C08939=1023.663,350.015,-141.631,171.610,48.646,159.588
C08940=1023.670,350.262,-141.669,171.618,48.645,159.589
C08941=1023.678,350.509,-141.706,171.625,48.645,159.590
C08942=1023.686,350.757,-141.744,171.632,48.644,159.591
C08943=1023.693,350.988,-141.779,171.639,48.644,159.591
C08944=1023.700,351.219,-141.813,171.645,48.643,159.592
C08945=1023.707,351.450,-141.849,171.651,48.643,159.593
C08946=1023.714,351.682,-141.884,171.658,48.643,159.594
C08947=1023.722,351.913,-141.919,171.665,48.642,159.595
C08948=1023.729,352.145,-141.954,171.671,48.642,159.596
C08949=1023.736,352.376,-141.990,171.678,48.641,159.597
C08950=1023.744,352.607,-142.025,171.685,48.641,159.598
C08951=1023.752,352.855,-142.063,171.692,48.640,159.598
C08952=1023.759,353.101,-142.101,171.699,48.640,159.599
C08953=1023.767,353.348,-142.138,171.706,48.640,159.600
C08954=1023.775,353.595,-142.177,171.713,48.639,159.601
C08955=1023.783,353.843,-142.214,171.721,48.639,159.602
C08956=1023.792,354.089,-142.252,171.727,48.638,159.603
C08957=1023.799,354.337,-142.290,171.735,48.638,159.604
C08958=1023.806,354.583,-142.328,171.742,48.638,159.605
C08959=1023.814,354.831,-142.366,171.749,48.637,159.606
C08960=1023.823,355.077,-142.404,171.757,48.637,159.607
C08961=1023.831,355.324,-142.442,171.764,48.637,159.608
C08962=1023.838,355.572,-142.480,171.771,48.636,159.609
C08963=1023.846,355.819,-142.518,171.779,48.636,159.610
C08964=1023.854,356.065,-142.557,171.786,48.636,159.611
C08965=1023.861,356.312,-142.595,171.793,48.636,159.612
C08966=1023.869,356.560,-142.633,171.801,48.635,159.613
C08967=1023.877,356.806,-142.670,171.808,48.635,159.614
C08968=1023.885,357.053,-142.709,171.815,48.634,159.615
C08969=1023.894,357.300,-142.748,171.823,48.634,159.616
C08970=1023.901,357.547,-142.786,171.830,48.634,159.617
C08971=1023.909,357.794,-142.824,171.837,48.634,159.618
C08972=1023.917,358.040,-142.863,171.845,48.634,159.619
C08973=1023.925,358.288,-142.901,171.852,48.634,159.620
C08974=1023.933,358.535,-142.940,171.860,48.633,159.622
C08975=1023.941,358.781,-142.978,171.867,48.633,159.623
C08976=1023.950,359.028,-143.016,171.874,48.633,159.624
C08977=1023.957,359.275,-143.054,171.883,48.633,159.625
C08978=1023.965,359.522,-143.093,171.890,48.633,159.626
C08979=1023.973,359.769,-143.132,171.898,48.633,159.627
C08980=1023.981,360.016,-143.170,171.905,48.632,159.628
C08981=1023.989,360.262,-143.209,171.912,48.632,159.629
C08982=1023.998,360.510,-143.248,171.920,48.632,159.630
C08983=1024.005,360.757,-143.287,171.927,48.632,159.631
C08984=1024.013,361.003,-143.326,171.935,48.632,159.632
C08985=1024.021,361.250,-143.365,171.942,48.632,159.633
C08986=1024.029,361.497,-143.403,171.950,48.632,159.634
C08987=1024.037,361.743,-143.442,171.958,48.632,159.636
C08988=1024.044,361.991,-143.481,171.966,48.632,159.637
C08989=1024.053,362.237,-143.521,171.973,48.632,159.638
C08990=1024.061,362.485,-143.559,171.981,48.632,159.639
C08991=1024.070,362.731,-143.599,171.988,48.632,159.640
C08992=1024.077,362.978,-143.637,171.997,48.632,159.641
C08993=1024.085,363.225,-143.677,172.004,48.633,159.643
C08994=1024.093,363.471,-143.716,172.012,48.632,159.644
C08995=1024.101,363.719,-143.755,172.019,48.633,159.645
C08996=1024.110,363.965,-143.794,172.027,48.632,159.646
C08997=1024.118,364.212,-143.833,172.035,48.633,159.647
C08998=1024.126,364.459,-143.873,172.043,48.633,159.648
C08999=1024.134,364.706,-143.912,172.050,48.633,159.650
C09000=1024.142,364.952,-143.951,172.058,48.633,159.651
C09001=1024.150,365.198,-143.990,172.066,48.633,159.652
C09002=1024.159,365.446,-144.029,172.074,48.634,159.653
C09003=1024.168,365.738,-144.076,172.084,48.633,159.655
C09004=1024.179,366.031,-144.123,172.093,48.633,159.656
C09005=1024.188,366.323,-144.169,172.103,48.634,159.657
C09006=1024.198,366.616,-144.216,172.111,48.634,159.659
C09007=1024.206,366.862,-144.256,172.120,48.634,159.660
C09008=1024.215,367.109,-144.295,172.128,48.635,159.661
C09009=1024.223,367.355,-144.334,172.136,48.635,159.663
C09010=1024.231,367.602,-144.374,172.144,48.635,159.664
C09011=1024.239,367.849,-144.413,172.152,48.635,159.665
C09012=1024.248,368.096,-144.453,172.159,48.636,159.666
C09013=1024.257,368.343,-144.492,172.168,48.636,159.668
C09014=1024.265,368.589,-144.533,172.176,48.636,159.669
C09015=1024.273,368.836,-144.572,172.184,48.637,159.670
C09016=1024.281,369.083,-144.612,172.192,48.637,159.671
C09017=1024.290,369.328,-144.652,172.200,48.637,159.673
C09018=1024.298,369.575,-144.692,172.208,48.638,159.674
C09019=1024.307,369.823,-144.732,172.216,48.638,159.675
C09020=1024.315,370.069,-144.773,172.225,48.638,159.676
C09021=1024.323,370.316,-144.812,172.232,48.639,159.678
C09022=1024.331,370.562,-144.853,172.241,48.640,159.679
C09023=1024.340,370.808,-144.892,172.249,48.640,159.681
C09024=1024.348,371.055,-144.933,172.258,48.640,159.682
C09025=1024.356,371.302,-144.973,172.265,48.641,159.683
C09026=1024.365,371.548,-145.013,172.274,48.641,159.685
C09027=1024.373,371.795,-145.054,172.282,48.642,159.686
C09028=1024.382,372.042,-145.093,172.291,48.642,159.687
C09029=1024.390,372.288,-145.134,172.299,48.643,159.689
C09030=1024.399,372.535,-145.174,172.307,48.643,159.690
C09031=1024.407,372.782,-145.214,172.316,48.644,159.691
C09032=1024.416,373.028,-145.254,172.324,48.644,159.693
C09033=1024.424,373.275,-145.295,172.333,48.645,159.694
C09034=1024.433,373.521,-145.335,172.341,48.645,159.695
C09035=1024.442,373.768,-145.376,172.349,48.646,159.697
C09036=1024.449,374.015,-145.416,172.357,48.647,159.698
C09037=1024.459,374.261,-145.457,172.366,48.647,159.700
C09038=1024.467,374.508,-145.497,172.375,48.648,159.701
C09039=1024.475,374.719,-145.532,172.382,48.648,159.702
C09040=1024.482,374.931,-145.567,172.389,48.649,159.703
C09041=1024.489,375.143,-145.602,172.397,48.649,159.705
C09042=1024.497,375.354,-145.637,172.404,48.650,159.706
C09043=1024.505,375.566,-145.671,172.412,48.650,159.707
C09044=1024.512,375.778,-145.706,172.419,48.651,159.708
C09045=1024.520,375.989,-145.741,172.426,48.651,159.710
C09046=1024.527,376.201,-145.776,172.434,48.652,159.711
C09047=1024.536,376.448,-145.817,172.443,48.653,159.712
C09048=1024.545,376.694,-145.858,172.451,48.653,159.714
C09049=1024.553,376.941,-145.899,172.459,48.655,159.715
C09050=1024.562,377.187,-145.939,172.468,48.655,159.717
C09051=1024.570,377.433,-145.981,172.477,48.656,159.718
C09052=1024.579,377.680,-146.022,172.485,48.657,159.720
C09053=1024.587,377.926,-146.063,172.494,48.658,159.721
C09054=1024.596,378.173,-146.104,172.503,48.659,159.723
C09055=1024.605,378.419,-146.146,172.512,48.659,159.724
C09056=1024.614,378.665,-146.186,172.520,48.660,159.726
C09057=1024.623,378.912,-146.228,172.529,48.661,159.727
C09058=1024.631,379.159,-146.269,172.538,48.662,159.729
C09059=1024.640,379.404,-146.310,172.547,48.663,159.730
C09060=1024.649,379.651,-146.352,172.555,48.663,159.732
C09061=1024.657,379.898,-146.393,172.565,48.665,159.734
C09062=1024.666,380.144,-146.435,172.574,48.665,159.735
C09063=1024.675,380.389,-146.475,172.583,48.666,159.737
C09064=1024.684,380.635,-146.517,172.592,48.667,159.738
C09065=1024.692,380.880,-146.559,172.601,48.668,159.740
C09066=1024.702,381.126,-146.600,172.610,48.669,159.741
C09067=1024.710,381.372,-146.641,172.618,48.670,159.743
C09068=1024.719,381.617,-146.682,172.628,48.671,159.745
C09069=1024.728,381.862,-146.724,172.636,48.672,159.746
C09070=1024.737,382.109,-146.766,172.645,48.673,159.748
C09071=1024.746,382.355,-146.807,172.654,48.674,159.749
C09072=1024.755,382.601,-146.849,172.664,48.675,159.751
C09073=1024.764,382.847,-146.890,172.673,48.676,159.753
C09074=1024.773,383.094,-146.932,172.682,48.677,159.754
C09075=1024.782,383.340,-146.974,172.691,48.678,159.756
C09076=1024.791,383.586,-147.015,172.700,48.680,159.757
C09077=1024.800,383.832,-147.058,172.710,48.680,159.759
C09078=1024.809,384.079,-147.100,172.719,48.681,159.761
C09079=1024.818,384.325,-147.141,172.728,48.683,159.762
C09080=1024.827,384.571,-147.183,172.738,48.684,159.764
C09081=1024.837,384.817,-147.225,172.747,48.685,159.766
C09082=1024.846,385.063,-147.267,172.756,48.686,159.767
C09083=1024.856,385.310,-147.309,172.765,48.687,159.769
C09084=1024.865,385.556,-147.351,172.775,48.688,159.771
C09085=1024.874,385.802,-147.393,172.784,48.690,159.773
C09086=1024.883,386.049,-147.435,172.793,48.691,159.774
C09087=1024.892,386.294,-147.477,172.803,48.692,159.776
C09088=1024.902,386.541,-147.520,172.812,48.693,159.778
C09089=1024.911,386.787,-147.561,172.822,48.695,159.780
C09090=1024.919,387.033,-147.605,172.832,48.696,159.781
C09091=1024.929,387.279,-147.647,172.841,48.697,159.783
C09092=1024.938,387.526,-147.689,172.851,48.698,159.785
C09093=1024.947,387.772,-147.731,172.860,48.700,159.786
C09094=1024.957,388.018,-147.774,172.869,48.701,159.788
C09095=1024.966,388.264,-147.817,172.880,48.702,159.790
C09096=1024.975,388.510,-147.860,172.889,48.704,159.792
C09097=1024.984,388.756,-147.902,172.899,48.705,159.794
C09098=1024.994,389.002,-147.945,172.908,48.706,159.795
C09099=1025.003,389.248,-147.987,172.919,48.708,159.797
C09100=1025.012,389.495,-148.031,172.928,48.709,159.799
C09101=1025.022,389.740,-148.073,172.938,48.710,159.801
C09102=1025.031,389.986,-148.116,172.947,48.712,159.803
C09103=1025.041,390.233,-148.158,172.958,48.713,159.805
C09104=1025.049,390.479,-148.201,172.967,48.715,159.806
C09105=1025.059,390.725,-148.244,172.977,48.716,159.808
C09106=1025.068,390.970,-148.287,172.987,48.718,159.810
C09107=1025.078,391.217,-148.331,172.997,48.720,159.812
C09108=1025.087,391.463,-148.373,173.006,48.721,159.814
C09109=1025.097,391.709,-148.417,173.017,48.723,159.816
C09110=1025.106,391.955,-148.460,173.026,48.725,159.818
C09111=1025.115,392.201,-148.503,173.036,48.726,159.820
C09112=1025.125,392.447,-148.546,173.047,48.727,159.821
C09113=1025.135,392.694,-148.589,173.056,48.729,159.823
C09114=1025.144,392.939,-148.633,173.067,48.731,159.825
C09115=1025.154,393.185,-148.675,173.077,48.732,159.827
C09116=1025.163,393.431,-148.720,173.087,48.734,159.829
C09117=1025.173,393.677,-148.763,173.097,48.736,159.831
C09118=1025.182,393.923,-148.806,173.108,48.738,159.833
C09119=1025.192,394.169,-148.850,173.117,48.739,159.835
C09120=1025.202,394.415,-148.894,173.128,48.741,159.837
C09121=1025.211,394.660,-148.937,173.138,48.743,159.839
C09122=1025.221,394.906,-148.981,173.147,48.745,159.841
C09123=1025.232,395.188,-149.030,173.159,48.746,159.843
C09124=1025.242,395.469,-149.081,173.171,48.748,159.846
C09125=1025.254,395.750,-149.131,173.183,48.751,159.848
C09126=1025.265,396.031,-149.181,173.195,48.753,159.850
C09127=1025.274,396.277,-149.225,173.206,48.754,159.852
C09128=1025.284,396.523,-149.268,173.216,48.756,159.855
C09129=1025.294,396.769,-149.312,173.227,48.758,159.856
C09130=1025.304,397.015,-149.356,173.236,48.760,159.858
C09131=1025.313,397.261,-149.400,173.247,48.762,159.861
C09132=1025.324,397.507,-149.444,173.258,48.763,159.863
C09133=1025.333,397.752,-149.488,173.269,48.766,159.865
C09134=1025.343,397.998,-149.532,173.279,48.767,159.867
C09135=1025.353,398.244,-149.576,173.290,48.769,159.869
C09136=1025.363,398.490,-149.621,173.301,48.771,159.871
C09137=1025.373,398.735,-149.664,173.311,48.773,159.873
C09138=1025.383,398.982,-149.709,173.322,48.775,159.875
C09139=1025.392,399.228,-149.754,173.333,48.777,159.878
C09140=1025.403,399.473,-149.798,173.343,48.779,159.880
C09141=1025.412,399.719,-149.842,173.354,48.781,159.882
C09142=1025.422,399.965,-149.887,173.365,48.783,159.884
C09143=1025.432,400.210,-149.932,173.376,48.785,159.886
C09144=1025.443,400.456,-149.976,173.387,48.787,159.888
C09145=1025.452,400.702,-150.020,173.397,48.789,159.891
C09146=1025.462,400.948,-150.065,173.408,48.792,159.893
C09147=1025.472,401.193,-150.110,173.419,48.794,159.895
C09148=1025.483,401.439,-150.155,173.430,48.796,159.897
C09149=1025.492,401.685,-150.199,173.441,48.798,159.899
C09150=1025.502,401.930,-150.244,173.452,48.800,159.902
C09151=1025.512,402.176,-150.289,173.463,48.803,159.904
C09152=1025.522,402.422,-150.334,173.475,48.804,159.906
C09153=1025.532,402.667,-150.379,173.485,48.807,159.908
C09154=1025.542,402.914,-150.424,173.497,48.809,159.911
C09155=1025.552,403.159,-150.470,173.508,48.811,159.913
C09156=1025.562,403.405,-150.515,173.518,48.813,159.915
C09157=1025.572,403.650,-150.560,173.531,48.816,159.918
C09158=1025.582,403.896,-150.605,173.541,48.818,159.920
C09159=1025.593,404.141,-150.650,173.553,48.821,159.922
C09160=1025.604,404.387,-150.695,173.563,48.823,159.924
C09161=1025.614,404.632,-150.741,173.576,48.825,159.927
C09162=1025.624,404.878,-150.786,173.586,48.827,159.929
C09163=1025.634,405.123,-150.831,173.598,48.830,159.932
C09164=1025.644,405.369,-150.877,173.610,48.832,159.934
C09165=1025.655,405.615,-150.922,173.621,48.835,159.936
C09166=1025.665,405.861,-150.967,173.632,48.837,159.939
C09167=1025.675,406.106,-151.013,173.644,48.839,159.941
C09168=1025.686,406.352,-151.059,173.655,48.842,159.944
C09169=1025.696,406.597,-151.104,173.668,48.844,159.946
C09170=1025.706,406.843,-151.150,173.679,48.847,159.948
C09171=1025.717,407.088,-151.196,173.690,48.850,159.951
C09172=1025.727,407.334,-151.242,173.702,48.852,159.953
C09173=1025.738,407.580,-151.288,173.713,48.854,159.956
C09174=1025.749,407.825,-151.333,173.726,48.857,159.958
C09175=1025.759,408.070,-151.379,173.738,48.859,159.961
C09176=1025.770,408.315,-151.424,173.749,48.862,159.963
C09177=1025.781,408.561,-151.470,173.761,48.864,159.966
C09178=1025.791,408.807,-151.516,173.772,48.867,159.968
C09179=1025.802,409.052,-151.562,173.785,48.870,159.971
C09180=1025.813,409.299,-151.608,173.796,48.872,159.973
C09181=1025.824,409.544,-151.654,173.808,48.874,159.976
C09182=1025.834,409.790,-151.700,173.821,48.877,159.978
C09183=1025.847,410.093,-151.758,173.835,48.881,159.981
C09184=1025.860,410.397,-151.815,173.850,48.884,159.985
C09185=1025.874,410.700,-151.872,173.865,48.887,159.988
C09186=1025.887,411.004,-151.931,173.881,48.891,159.991
C09187=1025.897,411.250,-151.977,173.893,48.893,159.994
C09188=1025.909,411.495,-152.023,173.905,48.897,159.996
C09189=1025.919,411.741,-152.070,173.917,48.899,159.999
C09190=1025.929,411.986,-152.117,173.930,48.902,160.002
C09191=1025.940,412.231,-152.163,173.942,48.905,160.004
C09192=1025.951,412.476,-152.210,173.954,48.908,160.007
C09193=1025.962,412.722,-152.257,173.966,48.911,160.010
C09194=1025.973,412.968,-152.303,173.979,48.913,160.012
C09195=1025.984,413.213,-152.350,173.991,48.916,160.015
C09196=1025.995,413.458,-152.397,174.004,48.919,160.018
C09197=1026.005,413.704,-152.444,174.017,48.922,160.020
C09198=1026.017,413.949,-152.491,174.029,48.925,160.023
C09199=1026.028,414.194,-152.538,174.042,48.928,160.026
C09200=1026.039,414.440,-152.586,174.055,48.931,160.029
C09201=1026.050,414.685,-152.633,174.067,48.934,160.031
C09202=1026.061,414.930,-152.680,174.080,48.936,160.034
C09203=1026.072,415.175,-152.726,174.093,48.940,160.037
C09204=1026.083,415.421,-152.774,174.105,48.943,160.040
C09205=1026.094,415.666,-152.821,174.118,48.946,160.043
C09206=1026.106,415.911,-152.868,174.131,48.949,160.045
C09207=1026.117,416.157,-152.917,174.145,48.952,160.048
C09208=1026.128,416.402,-152.963,174.157,48.955,160.051
C09209=1026.139,416.647,-153.011,174.170,48.958,160.054
C09210=1026.150,416.891,-153.059,174.183,48.961,160.057
C09211=1026.161,417.137,-153.106,174.196,48.965,160.060
C09212=1026.173,417.382,-153.154,174.209,48.967,160.062
C09213=1026.184,417.628,-153.202,174.223,48.970,160.065
C09214=1026.195,417.872,-153.250,174.236,48.974,160.068
C09215=1026.206,418.118,-153.297,174.249,48.977,160.071
C09216=1026.217,418.363,-153.346,174.262,48.980,160.074
C09217=1026.229,418.608,-153.393,174.275,48.983,160.077
C09218=1026.240,418.854,-153.442,174.288,48.987,160.080
C09219=1026.252,419.099,-153.489,174.303,48.990,160.083
C09220=1026.263,419.344,-153.538,174.316,48.994,160.086
C09221=1026.275,419.589,-153.586,174.329,48.997,160.089
C09222=1026.286,419.834,-153.634,174.343,49.000,160.092
C09223=1026.298,420.079,-153.682,174.356,49.004,160.095
C09224=1026.309,420.324,-153.730,174.370,49.007,160.098
C09225=1026.321,420.569,-153.779,174.383,49.011,160.101
C09226=1026.332,420.814,-153.827,174.397,49.014,160.104
C09227=1026.344,421.059,-153.875,174.411,49.017,160.107
C09228=1026.356,421.304,-153.924,174.424,49.020,160.110
C09229=1026.367,421.549,-153.972,174.439,49.024,160.114
C09230=1026.379,421.794,-154.020,174.452,49.027,160.117
C09231=1026.391,422.039,-154.070,174.466,49.031,160.120
C09232=1026.403,422.284,-154.118,174.480,49.034,160.123
C09233=1026.414,422.529,-154.167,174.494,49.038,160.126
C09234=1026.426,422.774,-154.216,174.508,49.042,160.129
C09235=1026.438,423.019,-154.265,174.522,49.045,160.132
C09236=1026.450,423.264,-154.313,174.536,49.049,160.136
C09237=1026.461,423.508,-154.362,174.550,49.052,160.139
C09238=1026.473,423.754,-154.412,174.564,49.056,160.142
C09239=1026.485,423.999,-154.461,174.578,49.059,160.145
C09240=1026.497,424.244,-154.510,174.593,49.063,160.148
C09241=1026.509,424.488,-154.559,174.607,49.067,160.152
C09242=1026.521,424.734,-154.608,174.622,49.070,160.155
C09243=1026.536,425.048,-154.672,174.641,49.075,160.159
C09244=1026.551,425.362,-154.735,174.658,49.080,160.164
C09245=1026.567,425.676,-154.798,174.677,49.085,160.168
C09246=1026.582,425.990,-154.861,174.696,49.090,160.172
C09247=1026.594,426.236,-154.911,174.711,49.094,160.175
C09248=1026.607,426.480,-154.961,174.725,49.098,160.179
C09249=1026.618,426.725,-155.010,174.740,49.101,160.182
C09250=1026.630,426.970,-155.060,174.755,49.105,160.186
C09251=1026.643,427.215,-155.110,174.770,49.109,160.189
C09252=1026.655,427.460,-155.160,174.785,49.113,160.192
C09253=1026.667,427.704,-155.210,174.799,49.117,160.196
C09254=1026.679,427.949,-155.260,174.814,49.121,160.199
C09255=1026.691,428.193,-155.310,174.830,49.124,160.203
C09256=1026.704,428.438,-155.360,174.845,49.128,160.206
C09257=1026.716,428.683,-155.410,174.860,49.133,160.210
C09258=1026.728,428.928,-155.460,174.875,49.136,160.213
C09259=1026.740,429.172,-155.510,174.890,49.140,160.217
C09260=1026.752,429.417,-155.560,174.905,49.145,160.220
C09261=1026.765,429.661,-155.611,174.921,49.148,160.224
C09262=1026.777,429.906,-155.661,174.936,49.153,160.228
C09263=1026.790,430.151,-155.712,174.952,49.156,160.231
C09264=1026.803,430.396,-155.762,174.967,49.161,160.235
C09265=1026.815,430.640,-155.813,174.983,49.165,160.238
C09266=1026.828,430.885,-155.863,174.998,49.169,160.242
C09267=1026.840,431.129,-155.914,175.014,49.173,160.246
C09268=1026.852,431.374,-155.964,175.030,49.177,160.249
C09269=1026.866,431.619,-156.015,175.046,49.181,160.253
C09270=1026.878,431.863,-156.066,175.061,49.186,160.257
C09271=1026.891,432.107,-156.117,175.077,49.190,160.260
C09272=1026.903,432.352,-156.167,175.093,49.194,160.264
C09273=1026.917,432.596,-156.218,175.109,49.198,160.268
C09274=1026.930,432.841,-156.269,175.124,49.202,160.272
C09275=1026.943,433.085,-156.320,175.141,49.207,160.275
C09276=1026.955,433.330,-156.371,175.157,49.211,160.279
C09277=1026.968,433.574,-156.423,175.173,49.215,160.283
C09278=1026.981,433.818,-156.474,175.189,49.220,160.287
C09279=1026.994,434.063,-156.525,175.205,49.224,160.291
C09280=1027.007,434.307,-156.577,175.222,49.228,160.295
C09281=1027.020,434.552,-156.628,175.238,49.233,160.298
C09282=1027.033,434.796,-156.680,175.255,49.238,160.302
C09283=1027.046,435.041,-156.731,175.271,49.242,160.306
C09284=1027.059,435.285,-156.783,175.287,49.246,160.310
C09285=1027.072,435.529,-156.834,175.304,49.251,160.314
C09286=1027.085,435.774,-156.886,175.321,49.255,160.318
C09287=1027.098,436.018,-156.938,175.338,49.260,160.322
C09288=1027.111,436.262,-156.990,175.354,49.264,160.326
C09289=1027.125,436.506,-157.042,175.371,49.269,160.330
C09290=1027.138,436.750,-157.094,175.388,49.274,160.334
C09291=1027.151,436.995,-157.146,175.405,49.278,160.338
C09292=1027.165,437.239,-157.198,175.421,49.283,160.342
C09293=1027.177,437.484,-157.250,175.439,49.287,160.346
C09294=1027.191,437.728,-157.302,175.456,49.292,160.350
C09295=1027.205,437.972,-157.355,175.473,49.297,160.354
C09296=1027.218,438.216,-157.407,175.490,49.302,160.359
C09297=1027.231,438.460,-157.459,175.508,49.306,160.363
C09298=1027.245,438.704,-157.512,175.525,49.311,160.367
C09299=1027.258,438.948,-157.564,175.543,49.316,160.371
C09300=1027.272,439.192,-157.617,175.560,49.320,160.375
C09301=1027.285,439.436,-157.669,175.577,49.325,160.379
C09302=1027.298,439.681,-157.722,175.595,49.330,160.384
C09303=1027.312,439.917,-157.774,175.613,49.335,160.388
C09304=1027.325,440.154,-157.825,175.630,49.340,160.392
C09305=1027.339,440.391,-157.876,175.646,49.344,160.396
C09306=1027.352,440.628,-157.928,175.664,49.349,160.400
C09307=1027.365,440.865,-157.978,175.682,49.353,160.405
C09308=1027.379,441.102,-158.031,175.699,49.358,160.409
C09309=1027.392,441.338,-158.082,175.717,49.363,160.413
C09310=1027.405,441.576,-158.133,175.734,49.368,160.417
C09311=1027.419,441.819,-158.187,175.752,49.373,160.422
C09312=1027.434,442.063,-158.240,175.771,49.378,160.426
C09313=1027.447,442.307,-158.293,175.789,49.383,160.431
C09314=1027.462,442.551,-158.347,175.807,49.388,160.435
C09315=1027.476,442.794,-158.400,175.825,49.393,160.439
C09316=1027.491,443.037,-158.453,175.844,49.398,160.444
C09317=1027.505,443.280,-158.505,175.863,49.403,160.448
C09318=1027.520,443.524,-158.557,175.881,49.408,160.453
C09319=1027.537,443.767,-158.608,175.900,49.412,160.457
C09320=1027.554,444.011,-158.659,175.918,49.417,160.461
C09321=1027.570,444.254,-158.711,175.937,49.422,160.466
C09322=1027.588,444.499,-158.761,175.956,49.426,160.470
C09323=1027.605,444.742,-158.811,175.975,49.430,160.475
C09324=1027.624,444.987,-158.860,175.994,49.435,160.479
C09325=1027.642,445.231,-158.910,176.014,49.439,160.484
C09326=1027.661,445.475,-158.959,176.033,49.443,160.488
C09327=1027.681,445.719,-159.007,176.052,49.448,160.492
C09328=1027.701,445.963,-159.056,176.072,49.451,160.497
C09329=1027.722,446.207,-159.103,176.092,49.455,160.501
C09330=1027.743,446.451,-159.150,176.111,49.460,160.506
C09331=1027.764,446.696,-159.197,176.131,49.463,160.510
C09332=1027.787,446.941,-159.243,176.151,49.467,160.514
C09333=1027.808,447.185,-159.289,176.171,49.471,160.519
C09334=1027.832,447.430,-159.336,176.190,49.474,160.523
C09335=1027.855,447.674,-159.381,176.211,49.478,160.527
C09336=1027.879,447.919,-159.425,176.231,49.482,160.532
C09337=1027.903,448.164,-159.470,176.252,49.485,160.536
C09338=1027.928,448.409,-159.514,176.272,49.489,160.540
C09339=1027.953,448.654,-159.557,176.292,49.492,160.545
C09340=1027.979,448.899,-159.601,176.313,49.495,160.549
C09341=1028.005,449.144,-159.644,176.333,49.498,160.553
C09342=1028.032,449.389,-159.687,176.354,49.501,160.558
C09343=1028.059,449.635,-159.728,176.375,49.504,160.562
C09344=1028.087,449.880,-159.770,176.396,49.508,160.566
C09345=1028.115,450.125,-159.811,176.416,49.511,160.571
C09346=1028.143,450.371,-159.852,176.438,49.514,160.575
C09347=1028.172,450.616,-159.893,176.459,49.517,160.579
C09348=1028.201,450.861,-159.933,176.480,49.519,160.583
C09349=1028.231,451.106,-159.973,176.502,49.522,160.588
C09350=1028.262,451.352,-160.012,176.522,49.525,160.592
C09351=1028.293,451.598,-160.051,176.544,49.528,160.597
C09352=1028.324,451.844,-160.089,176.566,49.530,160.601
C09353=1028.356,452.089,-160.127,176.588,49.532,160.605
C09354=1028.388,452.334,-160.165,176.610,49.535,160.609
C09355=1028.421,452.580,-160.203,176.631,49.537,160.614
C09356=1028.454,452.826,-160.240,176.653,49.540,160.618
C09357=1028.488,453.072,-160.276,176.675,49.542,160.622
C09358=1028.522,453.317,-160.313,176.697,49.544,160.627
C09359=1028.557,453.564,-160.348,176.720,49.546,160.631
C09360=1028.592,453.809,-160.383,176.743,49.549,160.635
C09361=1028.627,454.055,-160.418,176.765,49.550,160.639
C09362=1028.664,454.300,-160.453,176.787,49.553,160.644
C09363=1028.387,454.375,-160.789,176.789,49.613,160.664
C09364=1028.352,454.130,-160.755,176.767,49.612,160.659
C09365=1028.316,453.885,-160.720,176.744,49.610,160.655
C09366=1028.281,453.639,-160.684,176.722,49.608,160.651
C09367=1028.246,453.392,-160.649,176.700,49.605,160.646
C09368=1028.211,453.147,-160.613,176.678,49.603,160.642
C09369=1028.177,452.902,-160.577,176.656,49.601,160.638
C09370=1028.144,452.655,-160.540,176.633,49.599,160.633
C09371=1028.112,452.410,-160.503,176.612,49.597,160.629
C09372=1028.065,452.058,-160.449,176.580,49.594,160.623
C09373=1028.020,451.706,-160.394,176.549,49.590,160.617
C09374=1027.975,451.354,-160.339,176.518,49.586,160.611
C09375=1027.932,451.002,-160.282,176.487,49.582,160.604
C09376=1027.890,450.656,-160.225,176.457,49.579,160.598
C09377=1027.850,450.310,-160.169,176.427,49.575,160.592
C09378=1027.820,450.065,-160.128,176.407,49.572,160.588
C09379=1027.793,449.819,-160.087,176.385,49.569,160.584
C09380=1027.765,449.574,-160.044,176.364,49.566,160.580
C09381=1027.738,449.329,-160.003,176.344,49.563,160.575
C09382=1027.711,449.084,-159.960,176.323,49.560,160.571
C09383=1027.685,448.838,-159.917,176.303,49.557,160.567
C09384=1027.660,448.594,-159.874,176.282,49.554,160.562
C09385=1027.635,448.349,-159.830,176.261,49.551,160.558
C09386=1027.610,448.104,-159.786,176.241,49.547,160.554
C09387=1027.586,447.859,-159.741,176.221,49.544,160.549
C09388=1027.562,447.615,-159.697,176.201,49.540,160.545
C09389=1027.538,447.370,-159.651,176.180,49.537,160.541
C09390=1027.515,447.125,-159.605,176.160,49.533,160.536
C09391=1027.493,446.880,-159.560,176.140,49.529,160.532
C09392=1027.472,446.636,-159.513,176.121,49.526,160.528
C09393=1027.450,446.392,-159.466,176.101,49.522,160.523
C09394=1027.429,446.147,-159.418,176.081,49.518,160.519
C09395=1027.408,445.903,-159.371,176.062,49.514,160.514
C09396=1027.389,445.658,-159.323,176.042,49.510,160.510
C09397=1027.368,445.414,-159.274,176.022,49.506,160.506
C09398=1027.349,445.170,-159.226,176.003,49.502,160.501
C09399=1027.331,444.926,-159.176,175.984,49.498,160.497
C09400=1027.312,444.682,-159.126,175.965,49.493,160.493
C09401=1027.295,444.438,-159.076,175.946,49.489,160.488
C09402=1027.277,444.194,-159.026,175.927,49.485,160.484
C09403=1027.261,443.950,-158.975,175.908,49.480,160.479
C09404=1027.244,443.707,-158.924,175.889,49.476,160.475
C09405=1027.229,443.464,-158.872,175.870,49.471,160.470
C09406=1027.213,443.220,-158.820,175.852,49.467,160.466
C09407=1027.198,442.976,-158.768,175.833,49.462,160.462
C09408=1027.183,442.733,-158.714,175.814,49.457,160.457
C09409=1027.169,442.491,-158.662,175.796,49.452,160.453
C09410=1027.155,442.247,-158.608,175.778,49.447,160.448
C09411=1027.142,442.003,-158.556,175.759,49.442,160.444
C09412=1027.127,441.759,-158.502,175.741,49.437,160.439
C09413=1027.114,441.515,-158.449,175.723,49.433,160.435
C09414=1027.102,441.300,-158.402,175.706,49.428,160.431
C09415=1027.089,441.084,-158.356,175.691,49.424,160.427
C09416=1027.077,440.869,-158.309,175.675,49.420,160.423
C09417=1027.064,440.653,-158.262,175.660,49.415,160.420
C09418=1027.052,440.437,-158.215,175.643,49.411,160.416
C09419=1027.040,440.222,-158.168,175.628,49.407,160.412
C09420=1027.028,440.006,-158.121,175.612,49.403,160.408
C09421=1027.016,439.790,-158.075,175.597,49.399,160.405
C09422=1027.002,439.546,-158.022,175.579,49.394,160.400
C09423=1026.989,439.302,-157.969,175.561,49.389,160.396
C09424=1026.975,439.058,-157.917,175.543,49.385,160.392
C09425=1026.962,438.814,-157.864,175.526,49.380,160.388
C09426=1026.949,438.570,-157.811,175.509,49.375,160.384
C09427=1026.935,438.326,-157.759,175.491,49.371,160.379
C09428=1026.922,438.081,-157.707,175.474,49.366,160.375
C09429=1026.908,437.837,-157.654,175.456,49.362,160.371
C09430=1026.894,437.593,-157.602,175.440,49.356,160.367
C09431=1026.881,437.348,-157.550,175.422,49.352,160.363
C09432=1026.869,437.105,-157.498,175.406,49.348,160.359
C09433=1026.855,436.860,-157.446,175.388,49.343,160.355
C09434=1026.841,436.616,-157.394,175.371,49.339,160.351
C09435=1026.828,436.372,-157.342,175.354,49.334,160.347
C09436=1026.815,436.127,-157.290,175.337,49.330,160.343
C09437=1026.802,435.884,-157.238,175.321,49.325,160.339
C09438=1026.789,435.639,-157.186,175.304,49.321,160.335
C09439=1026.775,435.395,-157.135,175.287,49.317,160.331
C09440=1026.763,435.150,-157.083,175.271,49.313,160.327
C09441=1026.750,434.906,-157.031,175.254,49.308,160.323
C09442=1026.737,434.661,-156.980,175.238,49.303,160.319
C09443=1026.724,434.418,-156.929,175.222,49.299,160.315
C09444=1026.710,434.173,-156.877,175.205,49.295,160.311
C09445=1026.697,433.929,-156.825,175.189,49.291,160.308
C09446=1026.685,433.684,-156.774,175.172,49.286,160.304
C09447=1026.672,433.440,-156.723,175.156,49.282,160.300
C09448=1026.659,433.195,-156.672,175.140,49.278,160.296
C09449=1026.647,432.951,-156.621,175.124,49.273,160.292
C09450=1026.633,432.706,-156.570,175.108,49.269,160.289
C09451=1026.621,432.462,-156.519,175.092,49.265,160.285
C09452=1026.608,432.217,-156.468,175.075,49.261,160.281
C09453=1026.595,431.972,-156.417,175.059,49.257,160.277
C09454=1026.582,431.728,-156.366,175.043,49.253,160.274
C09455=1026.570,431.484,-156.316,175.029,49.249,160.270
C09456=1026.557,431.239,-156.265,175.012,49.245,160.267
C09457=1026.544,430.994,-156.214,174.996,49.241,160.263
C09458=1026.531,430.750,-156.164,174.981,49.236,160.259
C09459=1026.519,430.505,-156.113,174.966,49.233,160.256
C09460=1026.507,430.261,-156.063,174.949,49.229,160.252
C09461=1026.494,430.016,-156.013,174.935,49.225,160.248
C09462=1026.482,429.772,-155.962,174.919,49.221,160.245
C09463=1026.469,429.527,-155.912,174.904,49.217,160.241
C09464=1026.456,429.283,-155.862,174.888,49.213,160.238
C09465=1026.444,429.038,-155.812,174.873,49.209,160.234
C09466=1026.432,428.793,-155.762,174.857,49.205,160.231
C09467=1026.419,428.549,-155.711,174.843,49.201,160.227
C09468=1026.407,428.304,-155.661,174.828,49.197,160.224
C09469=1026.394,428.059,-155.611,174.812,49.194,160.220
C09470=1026.382,427.814,-155.561,174.797,49.190,160.217
C09471=1026.370,427.570,-155.511,174.783,49.186,160.213
C09472=1026.358,427.325,-155.462,174.767,49.182,160.210
C09473=1026.346,427.080,-155.412,174.752,49.178,160.206
C09474=1026.334,426.835,-155.362,174.738,49.174,160.203
C09475=1026.322,426.591,-155.312,174.723,49.171,160.200
C09476=1026.310,426.346,-155.262,174.708,49.167,160.196
C09477=1026.298,426.101,-155.212,174.693,49.163,160.193
C09478=1026.283,425.784,-155.148,174.674,49.158,160.188
C09479=1026.267,425.468,-155.084,174.655,49.154,160.184
C09480=1026.252,425.151,-155.021,174.636,49.149,160.180
C09481=1026.236,424.835,-154.957,174.618,49.144,160.176
C09482=1026.224,424.589,-154.908,174.603,49.141,160.172
C09483=1026.212,424.344,-154.859,174.589,49.137,160.169
C09484=1026.200,424.099,-154.810,174.575,49.134,160.166
C09485=1026.188,423.855,-154.760,174.561,49.130,160.163
C09486=1026.176,423.610,-154.711,174.546,49.126,160.159
C09487=1026.165,423.365,-154.662,174.532,49.123,160.156
C09488=1026.152,423.120,-154.613,174.518,49.120,160.153
C09489=1026.141,422.874,-154.565,174.504,49.116,160.150
C09490=1026.129,422.630,-154.516,174.489,49.113,160.147
C09491=1026.118,422.385,-154.467,174.476,49.109,160.144
C09492=1026.106,422.140,-154.418,174.462,49.105,160.140
C09493=1026.094,421.894,-154.370,174.448,49.103,160.137
C09494=1026.082,421.650,-154.321,174.434,49.099,160.134
C09495=1026.071,421.405,-154.272,174.420,49.095,160.131
C09496=1026.059,421.160,-154.224,174.406,49.092,160.128
C09497=1026.048,420.915,-154.176,174.392,49.089,160.125
C09498=1026.036,420.670,-154.127,174.379,49.085,160.122
C09499=1026.024,420.425,-154.079,174.365,49.083,160.119
C09500=1026.013,420.179,-154.031,174.352,49.079,160.116
C09501=1026.001,419.935,-153.982,174.338,49.076,160.113
C09502=1025.989,419.689,-153.934,174.325,49.072,160.110
C09503=1025.978,419.444,-153.886,174.311,49.069,160.107
C09504=1025.966,419.199,-153.838,174.298,49.066,160.104
C09505=1025.955,418.954,-153.791,174.284,49.063,160.101
C09506=1025.944,418.709,-153.742,174.271,49.060,160.098
C09507=1025.932,418.464,-153.695,174.257,49.057,160.095
C09508=1025.921,418.219,-153.646,174.244,49.054,160.092
C09509=1025.909,417.974,-153.599,174.231,49.050,160.089
C09510=1025.898,417.728,-153.550,174.217,49.047,160.086
C09511=1025.887,417.484,-153.503,174.204,49.044,160.083
C09512=1025.876,417.238,-153.455,174.191,49.041,160.080
C09513=1025.865,416.992,-153.407,174.177,49.038,160.077
C09514=1025.853,416.747,-153.359,174.164,49.035,160.074
C09515=1025.843,416.503,-153.312,174.151,49.031,160.072
C09516=1025.831,416.257,-153.265,174.139,49.029,160.069
C09517=1025.821,416.012,-153.217,174.125,49.026,160.066
C09518=1025.809,415.767,-153.170,174.112,49.023,160.063
C09519=1025.798,415.521,-153.123,174.099,49.020,160.060
C09520=1025.787,415.276,-153.074,174.087,49.017,160.058
C09521=1025.776,415.031,-153.028,174.074,49.014,160.055
C09522=1025.764,414.785,-152.981,174.061,49.011,160.052
C09523=1025.754,414.540,-152.934,174.049,49.008,160.049
C09524=1025.742,414.294,-152.887,174.036,49.005,160.046
C09525=1025.732,414.049,-152.840,174.022,49.003,160.044
C09526=1025.720,413.804,-152.792,174.010,49.000,160.041
C09527=1025.709,413.559,-152.745,173.997,48.997,160.038
C09528=1025.699,413.314,-152.698,173.985,48.994,160.036
C09529=1025.687,413.068,-152.652,173.972,48.991,160.033
C09530=1025.676,412.823,-152.606,173.961,48.988,160.030
C09531=1025.666,412.577,-152.558,173.948,48.985,160.027
C09532=1025.655,412.332,-152.511,173.935,48.983,160.025
C09533=1025.644,412.087,-152.465,173.923,48.980,160.022
C09534=1025.633,411.842,-152.418,173.911,48.977,160.020
C09535=1025.623,411.596,-152.372,173.898,48.975,160.017
C09536=1025.611,411.350,-152.325,173.885,48.972,160.014
C09537=1025.601,411.104,-152.279,173.874,48.969,160.012
C09538=1025.587,410.799,-152.221,173.859,48.966,160.008
C09539=1025.574,410.493,-152.162,173.844,48.962,160.005
C09540=1025.562,410.187,-152.105,173.828,48.959,160.002
C09541=1025.548,409.882,-152.047,173.813,48.956,159.999
C09542=1025.537,409.636,-152.001,173.801,48.954,159.996
C09543=1025.526,409.390,-151.954,173.789,48.951,159.994
C09544=1025.515,409.144,-151.909,173.777,48.949,159.991
C09545=1025.505,408.899,-151.863,173.765,48.946,159.989
C09546=1025.494,408.653,-151.817,173.753,48.943,159.986
C09547=1025.484,408.407,-151.771,173.741,48.941,159.984
C09548=1025.473,408.162,-151.725,173.729,48.939,159.981
C09549=1025.462,407.916,-151.679,173.718,48.936,159.979
C09550=1025.452,407.671,-151.634,173.706,48.934,159.976
C09551=1025.442,407.426,-151.588,173.693,48.931,159.974
C09552=1025.431,407.180,-151.542,173.682,48.929,159.971
C09553=1025.420,406.935,-151.496,173.670,48.926,159.969
C09554=1025.410,406.689,-151.450,173.659,48.924,159.967
C09555=1025.400,406.443,-151.405,173.647,48.922,159.964
C09556=1025.389,406.198,-151.360,173.636,48.919,159.962
C09557=1025.378,405.953,-151.314,173.623,48.917,159.959
C09558=1025.368,405.706,-151.269,173.613,48.915,159.957
C09559=1025.358,405.462,-151.223,173.601,48.912,159.955
C09560=1025.347,405.215,-151.178,173.589,48.910,159.952
C09561=1025.337,404.970,-151.132,173.578,48.908,159.950
C09562=1025.327,404.724,-151.087,173.566,48.906,159.947
C09563=1025.317,404.479,-151.041,173.555,48.904,159.945
C09564=1025.307,404.233,-150.996,173.544,48.901,159.943
C09565=1025.296,403.988,-150.951,173.532,48.899,159.940
C09566=1025.286,403.742,-150.906,173.521,48.896,159.938
C09567=1025.276,403.496,-150.861,173.510,48.894,159.936
C09568=1025.266,403.251,-150.815,173.499,48.892,159.934
C09569=1025.255,403.005,-150.770,173.487,48.890,159.931
C09570=1025.245,402.759,-150.726,173.476,48.888,159.929
C09571=1025.236,402.514,-150.681,173.465,48.886,159.927
C09572=1025.225,402.268,-150.636,173.455,48.884,159.925
C09573=1025.216,402.022,-150.591,173.443,48.882,159.922
C09574=1025.206,401.777,-150.546,173.432,48.880,159.920
C09575=1025.196,401.531,-150.501,173.421,48.877,159.918
C09576=1025.186,401.285,-150.456,173.410,48.875,159.915
C09577=1025.176,401.039,-150.411,173.399,48.873,159.913
C09578=1025.165,400.794,-150.366,173.388,48.871,159.911
C09579=1025.155,400.548,-150.322,173.378,48.869,159.909
C09580=1025.146,400.303,-150.277,173.366,48.867,159.907
C09581=1025.136,400.057,-150.233,173.355,48.865,159.905
C09582=1025.126,399.811,-150.188,173.344,48.863,159.902
C09583=1025.115,399.565,-150.143,173.333,48.861,159.900
C09584=1025.106,399.319,-150.099,173.323,48.860,159.898
C09585=1025.096,399.074,-150.055,173.312,48.857,159.896
C09586=1025.086,398.828,-150.011,173.301,48.855,159.894
C09587=1025.076,398.582,-149.966,173.290,48.854,159.892
C09588=1025.066,398.336,-149.923,173.280,48.852,159.889
C09589=1025.057,398.090,-149.878,173.269,48.850,159.887
C09590=1025.046,397.845,-149.834,173.258,48.848,159.885
C09591=1025.037,397.599,-149.790,173.248,48.846,159.883
C09592=1025.027,397.353,-149.747,173.237,48.844,159.881
C09593=1025.018,397.107,-149.702,173.226,48.843,159.879
C09594=1025.008,396.861,-149.658,173.216,48.841,159.877
C09595=1024.998,396.615,-149.614,173.205,48.839,159.875
C09596=1024.988,396.369,-149.570,173.196,48.837,159.873
C09597=1024.978,396.123,-149.526,173.185,48.836,159.871
C09598=1024.967,395.840,-149.476,173.173,48.834,159.869
C09599=1024.956,395.556,-149.425,173.161,48.831,159.866
C09600=1024.945,395.273,-149.375,173.149,48.830,159.864
C09601=1024.933,394.989,-149.325,173.137,48.828,159.862
C09602=1024.924,394.743,-149.281,173.127,48.826,159.860
C09603=1024.915,394.498,-149.238,173.116,48.825,159.858
C09604=1024.905,394.252,-149.194,173.106,48.823,159.856
C09605=1024.895,394.006,-149.150,173.096,48.821,159.854
C09606=1024.886,393.759,-149.107,173.086,48.819,159.852
C09607=1024.876,393.514,-149.064,173.076,48.818,159.850
C09608=1024.867,393.268,-149.020,173.065,48.816,159.848
C09609=1024.857,393.021,-148.977,173.056,48.815,159.846
C09610=1024.848,392.776,-148.934,173.045,48.813,159.844
C09611=1024.838,392.530,-148.890,173.035,48.812,159.842
C09612=1024.828,392.284,-148.847,173.024,48.810,159.840
C09613=1024.819,392.038,-148.804,173.015,48.809,159.838
C09614=1024.809,391.792,-148.761,173.005,48.807,159.836
C09615=1024.800,391.546,-148.718,172.995,48.806,159.835
C09616=1024.791,391.300,-148.675,172.985,48.804,159.833
C09617=1024.780,391.054,-148.631,172.975,48.803,159.831
C09618=1024.772,390.808,-148.588,172.966,48.802,159.829
C09619=1024.762,390.561,-148.546,172.955,48.800,159.827
C09620=1024.753,390.316,-148.503,172.945,48.799,159.825
C09621=1024.744,390.069,-148.460,172.936,48.798,159.823
C09622=1024.734,389.824,-148.417,172.925,48.796,159.821
C09623=1024.725,389.578,-148.374,172.916,48.795,159.820
C09624=1024.716,389.331,-148.331,172.906,48.794,159.818
C09625=1024.707,389.085,-148.288,172.897,48.792,159.816
C09626=1024.697,388.839,-148.246,172.887,48.791,159.814
C09627=1024.688,388.593,-148.204,172.877,48.789,159.812
C09628=1024.679,388.347,-148.161,172.867,48.788,159.811
C09629=1024.669,388.100,-148.118,172.858,48.786,159.809
C09630=1024.660,387.854,-148.076,172.848,48.785,159.807
C09631=1024.651,387.609,-148.033,172.839,48.784,159.805
C09632=1024.641,387.362,-147.990,172.828,48.783,159.803
C09633=1024.632,387.116,-147.949,172.819,48.782,159.802
C09634=1024.623,386.870,-147.906,172.810,48.780,159.800
C09635=1024.614,386.623,-147.863,172.800,48.779,159.798
C09636=1024.605,386.377,-147.821,172.791,48.778,159.797
C09637=1024.596,386.131,-147.779,172.781,48.777,159.795
C09638=1024.587,385.885,-147.737,172.772,48.776,159.793
C09639=1024.578,385.639,-147.695,172.763,48.775,159.792
C09640=1024.568,385.392,-147.652,172.753,48.774,159.790
C09641=1024.559,385.146,-147.611,172.744,48.772,159.788
C09642=1024.550,384.900,-147.568,172.734,48.772,159.786
C09643=1024.540,384.654,-147.527,172.725,48.771,159.785
C09644=1024.531,384.408,-147.485,172.716,48.769,159.783
C09645=1024.522,384.161,-147.444,172.706,48.769,159.781
C09646=1024.513,383.915,-147.401,172.697,48.767,159.780
C09647=1024.503,383.668,-147.359,172.688,48.767,159.778
C09648=1024.495,383.422,-147.318,172.679,48.765,159.776
C09649=1024.486,383.176,-147.276,172.669,48.764,159.775
C09650=1024.477,382.929,-147.234,172.660,48.764,159.773
C09651=1024.468,382.683,-147.192,172.651,48.763,159.772
C09652=1024.459,382.437,-147.151,172.642,48.761,159.770
C09653=1024.449,382.191,-147.110,172.632,48.761,159.768
C09654=1024.440,381.944,-147.068,172.623,48.760,159.767
C09655=1024.432,381.698,-147.026,172.614,48.759,159.765
C09656=1024.423,381.452,-146.985,172.606,48.758,159.764
C09657=1024.414,381.206,-146.943,172.595,48.757,159.762
C09658=1024.405,380.958,-146.902,172.587,48.756,159.760
C09659=1024.396,380.712,-146.860,172.578,48.755,159.759
C09660=1024.387,380.465,-146.819,172.569,48.755,159.757
C09661=1024.378,380.218,-146.777,172.560,48.753,159.756
C09662=1024.369,379.972,-146.736,172.551,48.752,159.754
C09663=1024.361,379.725,-146.695,172.542,48.752,159.753
C09664=1024.352,379.479,-146.653,172.533,48.751,159.751
C09665=1024.343,379.233,-146.611,172.524,48.750,159.750
C09666=1024.335,378.986,-146.570,172.515,48.750,159.748
C09667=1024.326,378.740,-146.529,172.506,48.749,159.746
C09668=1024.317,378.493,-146.488,172.498,48.748,159.745
C09669=1024.309,378.247,-146.446,172.489,48.747,159.743
C09670=1024.300,378.000,-146.406,172.480,48.746,159.742
C09671=1024.291,377.754,-146.364,172.471,48.746,159.740
C09672=1024.283,377.508,-146.324,172.463,48.745,159.739
C09673=1024.274,377.261,-146.282,172.454,48.744,159.737
C09674=1024.266,377.015,-146.241,172.445,48.743,159.736
C09675=1024.257,376.768,-146.200,172.437,48.743,159.735
C09676=1024.248,376.522,-146.159,172.428,48.742,159.733
C09677=1024.239,376.276,-146.119,172.419,48.741,159.732
C09678=1024.231,376.029,-146.078,172.410,48.741,159.730
C09679=1024.221,375.782,-146.037,172.402,48.740,159.729
C09680=1024.213,375.536,-145.996,172.393,48.740,159.727
C09681=1024.204,375.289,-145.956,172.385,48.739,159.726
C09682=1024.196,375.043,-145.915,172.376,48.739,159.724
C09683=1024.187,374.796,-145.875,172.367,48.738,159.723
C09684=1024.179,374.550,-145.834,172.359,48.738,159.722
C09685=1024.169,374.303,-145.794,172.350,48.737,159.720
C09686=1024.161,374.057,-145.753,172.342,48.737,159.719
C09687=1024.153,373.810,-145.712,172.333,48.736,159.717
C09688=1024.144,373.563,-145.673,172.324,48.736,159.716
C09689=1024.136,373.317,-145.632,172.317,48.735,159.715
C09690=1024.127,373.070,-145.592,172.308,48.735,159.713
C09691=1024.119,372.824,-145.551,172.300,48.734,159.712
C09692=1024.109,372.577,-145.511,172.291,48.734,159.711
C09693=1024.102,372.330,-145.471,172.283,48.734,159.709
C09694=1024.093,372.084,-145.431,172.274,48.733,159.708
C09695=1024.084,371.837,-145.390,172.266,48.733,159.706
C09696=1024.076,371.591,-145.351,172.258,48.732,159.705
C09697=1024.068,371.345,-145.310,172.250,48.732,159.704
C09698=1024.059,371.098,-145.271,172.241,48.731,159.702
C09699=1024.051,370.851,-145.230,172.233,48.731,159.701
C09700=1024.043,370.604,-145.190,172.224,48.731,159.700
C09701=1024.034,370.358,-145.150,172.217,48.730,159.699
C09702=1024.026,370.111,-145.110,172.208,48.730,159.697
C09703=1024.017,369.865,-145.069,172.200,48.730,159.696
C09704=1024.009,369.618,-145.029,172.192,48.729,159.695
C09705=1024.001,369.372,-144.989,172.183,48.729,159.693
C09706=1023.993,369.125,-144.950,172.176,48.729,159.692
C09707=1023.984,368.878,-144.910,172.167,48.728,159.691
C09708=1023.976,368.632,-144.870,172.159,48.728,159.689
C09709=1023.968,368.385,-144.830,172.151,48.728,159.688
C09710=1023.960,368.138,-144.790,172.143,48.727,159.687
C09711=1023.951,367.891,-144.751,172.135,48.727,159.686
C09712=1023.943,367.644,-144.711,172.127,48.728,159.685
C09713=1023.934,367.398,-144.672,172.119,48.727,159.683
C09714=1023.926,367.163,-144.634,172.111,48.727,159.682
C09715=1023.918,366.926,-144.596,172.104,48.727,159.681
C09716=1023.911,366.690,-144.559,172.095,48.727,159.680
C09717=1023.902,366.455,-144.521,172.088,48.727,159.679
C09718=1023.895,366.219,-144.484,172.081,48.726,159.677
C09719=1023.886,365.982,-144.446,172.073,48.727,159.676
C09720=1023.879,365.747,-144.408,172.066,48.727,159.675
C09721=1023.870,365.511,-144.371,172.058,48.726,159.674
C09722=1023.862,365.264,-144.331,172.050,48.727,159.673
C09723=1023.854,365.017,-144.291,172.042,48.726,159.672
C09724=1023.846,364.770,-144.253,172.035,48.726,159.671
C09725=1023.838,364.524,-144.214,172.026,48.726,159.669
C09726=1023.830,364.277,-144.174,172.018,48.726,159.668
C09727=1023.822,364.030,-144.136,172.011,48.726,159.667
C09728=1023.814,363.783,-144.096,172.003,48.726,159.666
C09729=1023.805,363.537,-144.057,171.995,48.726,159.665
C09730=1023.797,363.289,-144.018,171.987,48.726,159.663
C09731=1023.789,363.043,-143.979,171.979,48.727,159.662
C09732=1023.780,362.796,-143.939,171.972,48.726,159.661
C09733=1023.774,362.549,-143.901,171.964,48.726,159.660
C09734=1023.765,362.303,-143.861,171.957,48.726,159.659
C09735=1023.757,362.056,-143.823,171.948,48.726,159.658
C09736=1023.749,361.808,-143.784,171.941,48.726,159.657
C09737=1023.741,361.563,-143.745,171.933,48.727,159.655
C09738=1023.734,361.315,-143.706,171.926,48.727,159.654
C09739=1023.725,361.068,-143.666,171.918,48.727,159.653
C09740=1023.717,360.821,-143.628,171.910,48.726,159.652
C09741=1023.709,360.575,-143.590,171.902,48.727,159.651
C09742=1023.701,360.328,-143.550,171.895,48.727,159.650
C09743=1023.693,360.081,-143.512,171.887,48.727,159.649
C09744=1023.685,359.834,-143.473,171.880,48.727,159.648
C09745=1023.677,359.587,-143.435,171.872,48.728,159.647
C09746=1023.669,359.340,-143.396,171.865,48.728,159.646
C09747=1023.661,359.093,-143.358,171.857,48.728,159.645
C09748=1023.653,358.846,-143.319,171.850,48.728,159.643
C09749=1023.645,358.600,-143.280,171.842,48.728,159.642
C09750=1023.637,358.353,-143.242,171.835,48.728,159.641
C09751=1023.629,358.106,-143.203,171.828,48.729,159.641
C09752=1023.622,357.859,-143.166,171.820,48.730,159.639
C09753=1023.614,357.612,-143.127,171.813,48.730,159.638
C09754=1023.605,357.365,-143.089,171.805,48.730,159.637
C09755=1023.597,357.118,-143.051,171.798,48.730,159.636
C09756=1023.590,356.872,-143.013,171.790,48.731,159.635
C09757=1023.581,356.624,-142.974,171.783,48.731,159.634
C09758=1023.573,356.377,-142.935,171.776,48.731,159.633
C09759=1023.566,356.130,-142.898,171.768,48.732,159.632
C09760=1023.559,355.884,-142.860,171.761,48.732,159.631
C09761=1023.550,355.637,-142.822,171.753,48.732,159.630
C09762=1023.542,355.390,-142.783,171.746,48.733,159.629
C09763=1023.534,355.142,-142.745,171.739,48.733,159.628
C09764=1023.527,354.896,-142.707,171.731,48.733,159.627
C09765=1023.519,354.648,-142.669,171.724,48.734,159.626
C09766=1023.506,354.259,-142.609,171.713,48.735,159.625
C09767=1023.494,353.870,-142.550,171.702,48.735,159.623
C09768=1023.482,353.481,-142.491,171.690,48.736,159.622
C09769=1023.470,353.093,-142.430,171.679,48.737,159.620
C09770=1023.461,352.845,-142.393,171.672,48.737,159.619
C09771=1023.454,352.598,-142.356,171.664,48.738,159.618
C09772=1023.446,352.352,-142.318,171.657,48.738,159.617
C09773=1023.438,352.104,-142.280,171.650,48.739,159.617
C09774=1023.428,351.781,-142.230,171.640,48.740,159.615
C09775=1023.419,351.458,-142.182,171.631,48.741,159.614
C09776=1023.408,351.136,-142.133,171.622,48.741,159.613
C09777=1023.398,350.813,-142.083,171.613,48.742,159.612
C09778=1023.391,350.566,-142.046,171.605,48.743,159.611
C09779=1023.382,350.318,-142.008,171.599,48.744,159.610
C09780=1023.375,350.071,-141.971,171.592,48.744,159.609
C09781=1023.368,349.824,-141.933,171.585,48.745,159.608
C09782=1023.360,349.577,-141.897,171.577,48.745,159.607
C09783=1023.352,349.330,-141.859,171.570,48.746,159.606
C09784=1023.345,349.083,-141.821,171.564,48.747,159.606
C09785=1023.337,348.836,-141.785,171.557,48.747,159.605
C09786=1023.329,348.588,-141.747,171.550,48.748,159.604
C09787=1023.321,348.341,-141.710,171.543,48.749,159.603
C09788=1023.314,348.094,-141.672,171.536,48.750,159.602
C09789=1023.306,347.847,-141.635,171.529,48.750,159.601
C09790=1023.299,347.600,-141.598,171.522,48.751,159.600
C09791=1023.291,347.353,-141.561,171.515,48.752,159.599
C09792=1023.284,347.106,-141.524,171.508,48.752,159.599
C09793=1023.276,346.859,-141.487,171.502,48.754,159.598
C09794=1023.269,346.612,-141.450,171.495,48.754,159.597
C09795=1023.261,346.365,-141.413,171.488,48.755,159.596
C09796=1023.253,346.117,-141.376,171.480,48.756,159.595
C09797=1023.246,345.870,-141.339,171.474,48.757,159.595
C09798=1023.238,345.623,-141.302,171.467,48.758,159.594
C09799=1023.231,345.376,-141.265,171.461,48.759,159.593
C09800=1023.223,345.129,-141.228,171.454,48.759,159.592
C09801=1023.215,344.881,-141.192,171.447,48.760,159.591
C09802=1023.208,344.634,-141.154,171.440,48.761,159.591
C09803=1023.200,344.387,-141.118,171.433,48.762,159.590
C09804=1023.192,344.140,-141.081,171.426,48.763,159.589
C09805=1023.185,343.892,-141.044,171.420,48.764,159.588
C09806=1023.177,343.645,-141.008,171.413,48.765,159.587
C09807=1023.171,343.398,-140.971,171.407,48.766,159.587
C09808=1023.163,343.152,-140.934,171.400,48.766,159.586
C09809=1023.155,342.904,-140.898,171.393,48.767,159.585
C09810=1023.148,342.656,-140.861,171.386,48.769,159.584
C09811=1023.140,342.410,-140.824,171.379,48.769,159.584
C09812=1023.133,342.162,-140.788,171.373,48.771,159.583
C09813=1023.126,341.915,-140.752,171.366,48.771,159.582
C09814=1023.118,341.668,-140.715,171.360,48.773,159.581
C09815=1023.111,341.421,-140.678,171.353,48.774,159.581
C09816=1023.103,341.173,-140.642,171.347,48.774,159.580
C09817=1023.096,340.926,-140.605,171.340,48.776,159.579
C09818=1023.089,340.679,-140.569,171.334,48.776,159.578
C09819=1023.081,340.432,-140.533,171.327,48.778,159.578
C09820=1023.073,340.185,-140.496,171.321,48.779,159.577
C09821=1023.067,339.938,-140.460,171.313,48.780,159.576
C09822=1023.059,339.690,-140.424,171.307,48.781,159.576
C09823=1023.052,339.443,-140.387,171.300,48.782,159.575
C09824=1023.044,339.195,-140.351,171.294,48.783,159.574
C09825=1023.037,338.948,-140.315,171.287,48.784,159.573
C09826=1023.029,338.701,-140.279,171.281,48.785,159.573
C09827=1023.022,338.454,-140.243,171.274,48.787,159.572
C09828=1023.015,338.206,-140.208,171.268,48.788,159.572
C09829=1023.007,337.959,-140.172,171.262,48.789,159.571
C09830=1023.000,337.725,-140.137,171.255,48.791,159.570
C09831=1022.993,337.491,-140.103,171.250,48.791,159.570
C09832=1022.986,337.256,-140.069,171.244,48.793,159.569
C09833=1022.979,337.023,-140.035,171.237,48.794,159.568
C09834=1022.973,336.789,-140.002,171.231,48.795,159.568
C09835=1022.966,336.555,-139.967,171.225,48.796,159.567
C09836=1022.959,336.321,-139.933,171.219,48.797,159.566
C09837=1022.952,336.087,-139.900,171.213,48.799,159.566
C09838=1022.944,335.840,-139.863,171.206,48.800,159.565
C09839=1022.938,335.592,-139.828,171.200,48.801,159.565
C09840=1022.930,335.345,-139.792,171.194,48.803,159.564
C09841=1022.922,335.097,-139.756,171.187,48.804,159.563
C09842=1022.915,334.850,-139.721,171.181,48.805,159.563
C09843=1022.908,334.603,-139.685,171.174,48.806,159.562
C09844=1022.901,334.355,-139.649,171.168,48.808,159.561
C09845=1022.894,334.108,-139.614,171.162,48.809,159.561
C09846=1022.886,333.861,-139.577,171.155,48.810,159.560
C09847=1022.879,333.614,-139.542,171.150,48.811,159.559
C09848=1022.872,333.366,-139.506,171.144,48.813,159.559
C09849=1022.865,333.119,-139.471,171.138,48.814,159.558
C09850=1022.858,332.871,-139.435,171.131,48.815,159.558
C09851=1022.851,332.624,-139.399,171.125,48.817,159.557
C09852=1022.844,332.377,-139.364,171.119,48.819,159.557
C09853=1022.836,332.129,-139.329,171.112,48.820,159.556
C09854=1022.829,331.882,-139.294,171.106,48.821,159.555
C09855=1022.821,331.634,-139.258,171.100,48.823,159.555
C09856=1022.815,331.387,-139.223,171.094,48.824,159.554
C09857=1022.808,331.139,-139.188,171.087,48.825,159.553
C09858=1022.800,330.891,-139.153,171.081,48.827,159.553
C09859=1022.793,330.645,-139.117,171.075,48.829,159.552
C09860=1022.786,330.397,-139.082,171.069,48.831,159.552
C09861=1022.778,330.149,-139.046,171.062,48.832,159.551
C09862=1022.771,329.902,-139.012,171.056,48.834,159.551
C09863=1022.764,329.655,-138.977,171.050,48.835,159.550
C09864=1022.757,329.408,-138.942,171.044,48.837,159.550
C09865=1022.750,329.159,-138.906,171.038,48.838,159.549
C09866=1022.743,328.912,-138.872,171.032,48.840,159.549
C09867=1022.736,328.665,-138.836,171.026,48.841,159.548
C09868=1022.729,328.418,-138.801,171.020,48.843,159.548
C09869=1022.722,328.170,-138.766,171.014,48.844,159.547
C09870=1022.714,327.923,-138.731,171.008,48.846,159.546
C09871=1022.707,327.675,-138.696,171.001,48.847,159.546
C09872=1022.701,327.428,-138.661,170.995,48.849,159.545
C09873=1022.694,327.180,-138.626,170.989,48.851,159.545
C09874=1022.687,326.933,-138.591,170.983,48.852,159.544
C09875=1022.679,326.685,-138.556,170.978,48.854,159.544
C09876=1022.672,326.438,-138.522,170.972,48.856,159.543
C09877=1022.664,326.191,-138.487,170.966,48.858,159.543
C09878=1022.657,325.943,-138.452,170.960,48.859,159.542
C09879=1022.650,325.696,-138.418,170.953,48.861,159.542
C09880=1022.643,325.449,-138.384,170.947,48.863,159.541
C09881=1022.635,325.200,-138.348,170.941,48.864,159.541
C09882=1022.628,324.953,-138.315,170.935,48.866,159.540
C09883=1022.621,324.706,-138.280,170.929,48.868,159.540
C09884=1022.614,324.458,-138.246,170.923,48.870,159.539
C09885=1022.607,324.211,-138.211,170.917,48.872,159.539
C09886=1022.599,323.963,-138.177,170.911,48.874,159.539
C09887=1022.593,323.716,-138.142,170.906,48.876,159.538
C09888=1022.586,323.468,-138.108,170.900,48.877,159.538
C09889=1022.578,323.221,-138.074,170.894,48.879,159.537
C09890=1022.571,322.985,-138.041,170.888,48.881,159.537
C09891=1022.564,322.748,-138.009,170.883,48.883,159.536
C09892=1022.558,322.512,-137.975,170.877,48.885,159.536
C09893=1022.551,322.276,-137.942,170.871,48.887,159.535
C09894=1022.545,322.039,-137.910,170.866,48.888,159.535
C09895=1022.538,321.802,-137.877,170.860,48.890,159.535
C09896=1022.531,321.566,-137.845,170.855,48.892,159.534
C09897=1022.524,321.331,-137.812,170.849,48.893,159.534
C09898=1022.517,321.083,-137.778,170.843,48.895,159.533
C09899=1022.510,320.835,-137.744,170.837,48.897,159.533
C09900=1022.503,320.587,-137.709,170.832,48.899,159.533
C09901=1022.496,320.340,-137.675,170.826,48.901,159.532
C09902=1022.488,320.092,-137.641,170.820,48.903,159.532
C09903=1022.483,319.845,-137.607,170.814,48.905,159.531
C09904=1022.475,319.597,-137.573,170.808,48.907,159.531
C09905=1022.468,319.350,-137.539,170.802,48.910,159.531
C09906=1022.461,319.103,-137.505,170.797,48.911,159.530
C09907=1022.454,318.855,-137.470,170.791,48.913,159.530
C09908=1022.447,318.607,-137.437,170.785,48.915,159.529
C09909=1022.440,318.360,-137.403,170.779,48.917,159.529
C09910=1022.434,318.112,-137.369,170.773,48.919,159.529
C09911=1022.427,317.864,-137.335,170.768,48.921,159.528
C09912=1022.420,317.617,-137.301,170.763,48.923,159.528
C09913=1022.412,317.369,-137.267,170.757,48.925,159.527
C09914=1022.407,317.122,-137.233,170.751,48.927,159.527
C09915=1022.399,316.874,-137.199,170.745,48.930,159.527
C09916=1022.392,316.626,-137.166,170.740,48.931,159.526
C09917=1022.386,316.379,-137.131,170.734,48.933,159.526
C09918=1022.379,316.132,-137.098,170.728,48.936,159.526
C09919=1022.372,315.884,-137.064,170.722,48.938,159.525
C09920=1022.365,315.636,-137.030,170.717,48.940,159.525
C09921=1022.359,315.389,-136.996,170.711,48.942,159.524
C09922=1022.352,315.141,-136.962,170.706,48.944,159.524
C09923=1022.344,314.894,-136.928,170.700,48.946,159.524
C09924=1022.339,314.646,-136.894,170.695,48.948,159.523
C09925=1022.331,314.399,-136.860,170.689,48.950,159.523
C09926=1022.324,314.150,-136.827,170.683,48.952,159.523
C09927=1022.318,313.903,-136.794,170.677,48.955,159.522
C09928=1022.311,313.655,-136.759,170.673,48.957,159.522
C09929=1022.305,313.408,-136.726,170.666,48.959,159.522
C09930=1022.298,313.161,-136.692,170.661,48.961,159.521
C09931=1022.291,312.913,-136.659,170.656,48.963,159.521
C09932=1022.285,312.665,-136.625,170.650,48.965,159.521
C09933=1022.278,312.417,-136.591,170.644,48.967,159.520
C09934=1022.271,312.170,-136.558,170.639,48.970,159.520
C09935=1022.264,311.922,-136.525,170.634,48.972,159.520
C09936=1022.258,311.675,-136.491,170.628,48.974,159.519
C09937=1022.251,311.427,-136.457,170.622,48.976,159.519
C09938=1022.245,311.180,-136.424,170.617,48.979,159.519
C09939=1022.238,310.932,-136.390,170.611,48.981,159.518
C09940=1022.232,310.684,-136.357,170.606,48.983,159.518
C09941=1022.225,310.437,-136.323,170.601,48.985,159.518
C09942=1022.218,310.189,-136.290,170.595,48.987,159.517
C09943=1022.212,309.942,-136.257,170.589,48.990,159.517
C09944=1022.204,309.694,-136.224,170.583,48.992,159.517
C09945=1022.198,309.447,-136.191,170.579,48.995,159.517
C09946=1022.191,309.199,-136.158,170.573,48.997,159.516
C09947=1022.184,308.951,-136.126,170.567,49.000,159.516
C09948=1022.177,308.703,-136.093,170.562,49.002,159.516
C09949=1022.170,308.456,-136.060,170.557,49.004,159.516
C09950=1022.163,308.222,-136.029,170.551,49.007,159.515
C09951=1022.157,307.988,-135.998,170.547,49.009,159.515
C09952=1022.151,307.754,-135.967,170.541,49.012,159.515
C09953=1022.144,307.520,-135.936,170.536,49.014,159.515
C09954=1022.137,307.287,-135.905,170.531,49.016,159.514
C09955=1022.131,307.053,-135.874,170.526,49.019,159.514
C09956=1022.124,306.820,-135.843,170.521,49.021,159.514
C09957=1022.118,306.586,-135.812,170.516,49.023,159.514
C09958=1022.111,306.338,-135.780,170.510,49.026,159.513
C09959=1022.104,306.090,-135.747,170.506,49.029,159.513
C09960=1022.097,305.843,-135.715,170.500,49.031,159.513
C09961=1022.091,305.595,-135.682,170.494,49.034,159.513
C09962=1022.084,305.347,-135.649,170.490,49.036,159.513
C09963=1022.077,305.100,-135.617,170.484,49.039,159.512
C09964=1022.071,304.852,-135.584,170.478,49.042,159.512
C09965=1022.064,304.604,-135.551,170.473,49.044,159.512
C09966=1022.057,304.356,-135.519,170.468,49.047,159.512
C09967=1022.051,304.109,-135.486,170.462,49.049,159.512
C09968=1022.043,303.861,-135.453,170.457,49.052,159.511
C09969=1022.037,303.613,-135.421,170.452,49.054,159.511
C09970=1022.030,303.366,-135.388,170.447,49.057,159.511
C09971=1022.023,303.118,-135.355,170.441,49.060,159.511
C09972=1022.017,302.869,-135.323,170.436,49.063,159.511
C09973=1022.010,302.622,-135.291,170.431,49.065,159.510
C09974=1022.003,302.375,-135.259,170.425,49.067,159.510
C09975=1021.997,302.127,-135.226,170.420,49.071,159.510
C09976=1021.989,301.879,-135.193,170.415,49.073,159.510
C09977=1021.983,301.631,-135.161,170.410,49.075,159.510
C09978=1021.977,301.383,-135.129,170.404,49.079,159.510
C09979=1021.970,301.136,-135.096,170.400,49.081,159.509
C09980=1021.964,300.888,-135.064,170.394,49.084,159.509
C09981=1021.957,300.640,-135.032,170.389,49.087,159.509
C09982=1021.950,300.392,-134.999,170.384,49.089,159.509
C09983=1021.944,300.145,-134.966,170.379,49.092,159.509
C09984=1021.937,299.897,-134.935,170.373,49.095,159.508
C09985=1021.931,299.649,-134.902,170.369,49.097,159.508
C09986=1021.924,299.402,-134.870,170.363,49.100,159.508
C09987=1021.918,299.154,-134.838,170.358,49.103,159.508
C09988=1021.911,298.905,-134.805,170.353,49.105,159.508
C09989=1021.904,298.657,-134.773,170.348,49.109,159.508
C09990=1021.898,298.410,-134.741,170.343,49.111,159.508
C09991=1021.891,298.162,-134.709,170.338,49.114,159.507
C09992=1021.885,297.914,-134.677,170.332,49.117,159.507
C09993=1021.879,297.667,-134.644,170.328,49.119,159.507
C09994=1021.872,297.419,-134.612,170.322,49.122,159.507
C09995=1021.866,297.171,-134.580,170.316,49.125,159.507
C09996=1021.859,296.923,-134.548,170.312,49.128,159.507
//INST
///DATE 2021/06/17 10:59
///ATTR SC,RW,RJ
////FRAME ROBOT
///GROUP1 RB1
NOP
MOVL C00000 V=800.0 PL=0
MOVL C00001 V=800.0 PL=0
MOVL C00002 V=800.0 PL=0
MOVL C00003 V=800.0 PL=0
MOVL C00004 V=800.0 PL=0
MOVL C00005 V=800.0 PL=0
MOVL C00006 V=800.0 PL=0
MOVL C00007 V=800.0 PL=0
MOVL C00008 V=800.0 PL=0
MOVL C00009 V=800.0 PL=0
MOVL C00010 V=800.0 PL=0
MOVL C00011 V=800.0 PL=0
MOVL C00012 V=800.0 PL=0
MOVL C00013 V=800.0 PL=0
MOVL C00014 V=800.0 PL=0
MOVL C00015 V=800.0 PL=0
MOVL C00016 V=800.0 PL=0
MOVL C00017 V=800.0 PL=0
MOVL C00018 V=800.0 PL=0
MOVL C00019 V=800.0 PL=0
MOVL C00020 V=800.0 PL=0
MOVL C00021 V=800.0 PL=0
MOVL C00022 V=800.0 PL=0
MOVL C00023 V=800.0 PL=0
MOVL C00024 V=800.0 PL=0
MOVL C00025 V=800.0 PL=0
MOVL C00026 V=800.0 PL=0
MOVL C00027 V=800.0 PL=0
MOVL C00028 V=800.0 PL=0
MOVL C00029 V=800.0 PL=0
MOVL C00030 V=800.0 PL=0
MOVL C00031 V=800.0 PL=0
MOVL C00032 V=800.0 PL=0
MOVL C00033 V=800.0 PL=0
MOVL C00034 V=800.0 PL=0
MOVL C00035 V=800.0 PL=0
MOVL C00036 V=800.0 PL=0
MOVL C00037 V=800.0 PL=0
MOVL C00038 V=800.0 PL=0
MOVL C00039 V=800.0 PL=0
MOVL C00040 V=800.0 PL=0
MOVL C00041 V=800.0 PL=0
MOVL C00042 V=800.0 PL=0
MOVL C00043 V=800.0 PL=0
MOVL C00044 V=800.0 PL=0
MOVL C00045 V=800.0 PL=0
MOVL C00046 V=800.0 PL=0
MOVL C00047 V=800.0 PL=0
MOVL C00048 V=800.0 PL=0
MOVL C00049 V=800.0 PL=0
MOVL C00050 V=800.0 PL=0
MOVL C00051 V=800.0 PL=0
MOVL C00052 V=800.0 PL=0
MOVL C00053 V=800.0 PL=0
MOVL C00054 V=800.0 PL=0
MOVL C00055 V=800.0 PL=0
MOVL C00056 V=800.0 PL=0
MOVL C00057 V=800.0 PL=0
MOVL C00058 V=800.0 PL=0
MOVL C00059 V=800.0 PL=0
MOVL C00060 V=800.0 PL=0
MOVL C00061 V=800.0 PL=0
MOVL C00062 V=800.0 PL=0
MOVL C00063 V=800.0 PL=0
MOVL C00064 V=800.0 PL=0
MOVL C00065 V=800.0 PL=0
MOVL C00066 V=800.0 PL=0
MOVL C00067 V=800.0 PL=0
MOVL C00068 V=800.0 PL=0
MOVL C00069 V=800.0 PL=0
MOVL C00070 V=800.0 PL=0
MOVL C00071 V=800.0 PL=0
MOVL C00072 V=800.0 PL=0
MOVL C00073 V=800.0 PL=0
MOVL C00074 V=800.0 PL=0
MOVL C00075 V=800.0 PL=0
MOVL C00076 V=800.0 PL=0
MOVL C00077 V=800.0 PL=0
MOVL C00078 V=800.0 PL=0
MOVL C00079 V=800.0 PL=0
MOVL C00080 V=800.0 PL=0
MOVL C00081 V=800.0 PL=0
MOVL C00082 V=800.0 PL=0
MOVL C00083 V=800.0 PL=0
MOVL C00084 V=800.0 PL=0
MOVL C00085 V=800.0 PL=0
MOVL C00086 V=800.0 PL=0
MOVL C00087 V=800.0 PL=0
MOVL C00088 V=800.0 PL=0
MOVL C00089 V=800.0 PL=0
MOVL C00090 V=800.0 PL=0
MOVL C00091 V=800.0 PL=0
MOVL C00092 V=800.0 PL=0
MOVL C00093 V=800.0 PL=0
MOVL C00094 V=800.0 PL=0
MOVL C00095 V=800.0 PL=0
MOVL C00096 V=800.0 PL=0
MOVL C00097 V=800.0 PL=0
MOVL C00098 V=800.0 PL=0
MOVL C00099 V=800.0 PL=0
MOVL C00100 V=800.0 PL=0
MOVL C00101 V=800.0 PL=0
MOVL C00102 V=800.0 PL=0
MOVL C00103 V=800.0 PL=0
MOVL C00104 V=800.0 PL=0
MOVL C00105 V=800.0 PL=0
MOVL C00106 V=800.0 PL=0
MOVL C00107 V=800.0 PL=0
MOVL C00108 V=800.0 PL=0
MOVL C00109 V=800.0 PL=0
MOVL C00110 V=800.0 PL=0
MOVL C00111 V=800.0 PL=0
MOVL C00112 V=800.0 PL=0
MOVL C00113 V=800.0 PL=0
MOVL C00114 V=800.0 PL=0
MOVL C00115 V=800.0 PL=0
MOVL C00116 V=800.0 PL=0
MOVL C00117 V=800.0 PL=0
MOVL C00118 V=800.0 PL=0
MOVL C00119 V=800.0 PL=0
MOVL C00120 V=800.0 PL=0
MOVL C00121 V=800.0 PL=0
MOVL C00122 V=800.0 PL=0
MOVL C00123 V=800.0 PL=0
MOVL C00124 V=800.0 PL=0
MOVL C00125 V=800.0 PL=0
MOVL C00126 V=800.0 PL=0
MOVL C00127 V=800.0 PL=0
MOVL C00128 V=800.0 PL=0
MOVL C00129 V=800.0 PL=0
MOVL C00130 V=800.0 PL=0
MOVL C00131 V=800.0 PL=0
MOVL C00132 V=800.0 PL=0
MOVL C00133 V=800.0 PL=0
MOVL C00134 V=800.0 PL=0
MOVL C00135 V=800.0 PL=0
MOVL C00136 V=800.0 PL=0
MOVL C00137 V=800.0 PL=0
MOVL C00138 V=800.0 PL=0
MOVL C00139 V=800.0 PL=0
MOVL C00140 V=800.0 PL=0
MOVL C00141 V=800.0 PL=0
MOVL C00142 V=800.0 PL=0
MOVL C00143 V=800.0 PL=0
MOVL C00144 V=800.0 PL=0
MOVL C00145 V=800.0 PL=0
MOVL C00146 V=800.0 PL=0
MOVL C00147 V=800.0 PL=0
MOVL C00148 V=800.0 PL=0
MOVL C00149 V=800.0 PL=0
MOVL C00150 V=800.0 PL=0
MOVL C00151 V=800.0 PL=0
MOVL C00152 V=800.0 PL=0
MOVL C00153 V=800.0 PL=0
MOVL C00154 V=800.0 PL=0
MOVL C00155 V=800.0 PL=0
MOVL C00156 V=800.0 PL=0
MOVL C00157 V=800.0 PL=0
MOVL C00158 V=800.0 PL=0
MOVL C00159 V=800.0 PL=0
MOVL C00160 V=800.0 PL=0
MOVL C00161 V=800.0 PL=0
MOVL C00162 V=800.0 PL=0
MOVL C00163 V=800.0 PL=0
MOVL C00164 V=800.0 PL=0
MOVL C00165 V=800.0 PL=0
MOVL C00166 V=800.0 PL=0
MOVL C00167 V=800.0 PL=0
MOVL C00168 V=800.0 PL=0
MOVL C00169 V=800.0 PL=0
MOVL C00170 V=800.0 PL=0
MOVL C00171 V=800.0 PL=0
MOVL C00172 V=800.0 PL=0
MOVL C00173 V=800.0 PL=0
MOVL C00174 V=800.0 PL=0
MOVL C00175 V=800.0 PL=0
MOVL C00176 V=800.0 PL=0
MOVL C00177 V=800.0 PL=0
MOVL C00178 V=800.0 PL=0
MOVL C00179 V=800.0 PL=0
MOVL C00180 V=800.0 PL=0
MOVL C00181 V=800.0 PL=0
MOVL C00182 V=800.0 PL=0
MOVL C00183 V=800.0 PL=0
MOVL C00184 V=800.0 PL=0
MOVL C00185 V=800.0 PL=0
MOVL C00186 V=800.0 PL=0
MOVL C00187 V=800.0 PL=0
MOVL C00188 V=800.0 PL=0
MOVL C00189 V=800.0 PL=0
MOVL C00190 V=800.0 PL=0
MOVL C00191 V=800.0 PL=0
MOVL C00192 V=800.0 PL=0
MOVL C00193 V=800.0 PL=0
MOVL C00194 V=800.0 PL=0
MOVL C00195 V=800.0 PL=0
MOVL C00196 V=800.0 PL=0
MOVL C00197 V=800.0 PL=0
MOVL C00198 V=800.0 PL=0
MOVL C00199 V=800.0 PL=0
MOVL C00200 V=800.0 PL=0
MOVL C00201 V=800.0 PL=0
MOVL C00202 V=800.0 PL=0
MOVL C00203 V=800.0 PL=0
MOVL C00204 V=800.0 PL=0
MOVL C00205 V=800.0 PL=0
MOVL C00206 V=800.0 PL=0
MOVL C00207 V=800.0 PL=0
MOVL C00208 V=800.0 PL=0
MOVL C00209 V=800.0 PL=0
MOVL C00210 V=800.0 PL=0
MOVL C00211 V=800.0 PL=0
MOVL C00212 V=800.0 PL=0
MOVL C00213 V=800.0 PL=0
MOVL C00214 V=800.0 PL=0
MOVL C00215 V=800.0 PL=0
MOVL C00216 V=800.0 PL=0
MOVL C00217 V=800.0 PL=0
MOVL C00218 V=800.0 PL=0
MOVL C00219 V=800.0 PL=0
MOVL C00220 V=800.0 PL=0
MOVL C00221 V=800.0 PL=0
MOVL C00222 V=800.0 PL=0
MOVL C00223 V=800.0 PL=0
MOVL C00224 V=800.0 PL=0
MOVL C00225 V=800.0 PL=0
MOVL C00226 V=800.0 PL=0
MOVL C00227 V=800.0 PL=0
MOVL C00228 V=800.0 PL=0
MOVL C00229 V=800.0 PL=0
MOVL C00230 V=800.0 PL=0
MOVL C00231 V=800.0 PL=0
MOVL C00232 V=800.0 PL=0
MOVL C00233 V=800.0 PL=0
MOVL C00234 V=800.0 PL=0
MOVL C00235 V=800.0 PL=0
MOVL C00236 V=800.0 PL=0
MOVL C00237 V=800.0 PL=0
MOVL C00238 V=800.0 PL=0
MOVL C00239 V=800.0 PL=0
MOVL C00240 V=800.0 PL=0
MOVL C00241 V=800.0 PL=0
MOVL C00242 V=800.0 PL=0
MOVL C00243 V=800.0 PL=0
MOVL C00244 V=800.0 PL=0
MOVL C00245 V=800.0 PL=0
MOVL C00246 V=800.0 PL=0
MOVL C00247 V=800.0 PL=0
MOVL C00248 V=800.0 PL=0
MOVL C00249 V=800.0 PL=0
MOVL C00250 V=800.0 PL=0
MOVL C00251 V=800.0 PL=0
MOVL C00252 V=800.0 PL=0
MOVL C00253 V=800.0 PL=0
MOVL C00254 V=800.0 PL=0
MOVL C00255 V=800.0 PL=0
MOVL C00256 V=800.0 PL=0
MOVL C00257 V=800.0 PL=0
MOVL C00258 V=800.0 PL=0
MOVL C00259 V=800.0 PL=0
MOVL C00260 V=800.0 PL=0
MOVL C00261 V=800.0 PL=0
MOVL C00262 V=800.0 PL=0
MOVL C00263 V=800.0 PL=0
MOVL C00264 V=800.0 PL=0
MOVL C00265 V=800.0 PL=0
MOVL C00266 V=800.0 PL=0
MOVL C00267 V=800.0 PL=0
MOVL C00268 V=800.0 PL=0
MOVL C00269 V=800.0 PL=0
MOVL C00270 V=800.0 PL=0
MOVL C00271 V=800.0 PL=0
MOVL C00272 V=800.0 PL=0
MOVL C00273 V=800.0 PL=0
MOVL C00274 V=800.0 PL=0
MOVL C00275 V=800.0 PL=0
MOVL C00276 V=800.0 PL=0
MOVL C00277 V=800.0 PL=0
MOVL C00278 V=800.0 PL=0
MOVL C00279 V=800.0 PL=0
MOVL C00280 V=800.0 PL=0
MOVL C00281 V=800.0 PL=0
MOVL C00282 V=800.0 PL=0
MOVL C00283 V=800.0 PL=0
MOVL C00284 V=800.0 PL=0
MOVL C00285 V=800.0 PL=0
MOVL C00286 V=800.0 PL=0
MOVL C00287 V=800.0 PL=0
MOVL C00288 V=800.0 PL=0
MOVL C00289 V=800.0 PL=0
MOVL C00290 V=800.0 PL=0
MOVL C00291 V=800.0 PL=0
MOVL C00292 V=800.0 PL=0
MOVL C00293 V=800.0 PL=0
MOVL C00294 V=800.0 PL=0
MOVL C00295 V=800.0 PL=0
MOVL C00296 V=800.0 PL=0
MOVL C00297 V=800.0 PL=0
MOVL C00298 V=800.0 PL=0
MOVL C00299 V=800.0 PL=0
MOVL C00300 V=800.0 PL=0
MOVL C00301 V=800.0 PL=0
MOVL C00302 V=800.0 PL=0
MOVL C00303 V=800.0 PL=0
MOVL C00304 V=800.0 PL=0
MOVL C00305 V=800.0 PL=0
MOVL C00306 V=800.0 PL=0
MOVL C00307 V=800.0 PL=0
MOVL C00308 V=800.0 PL=0
MOVL C00309 V=800.0 PL=0
MOVL C00310 V=800.0 PL=0
MOVL C00311 V=800.0 PL=0
MOVL C00312 V=800.0 PL=0
MOVL C00313 V=800.0 PL=0
MOVL C00314 V=800.0 PL=0
MOVL C00315 V=800.0 PL=0
MOVL C00316 V=800.0 PL=0
MOVL C00317 V=800.0 PL=0
MOVL C00318 V=800.0 PL=0
MOVL C00319 V=800.0 PL=0
MOVL C00320 V=800.0 PL=0
MOVL C00321 V=800.0 PL=0
MOVL C00322 V=800.0 PL=0
MOVL C00323 V=800.0 PL=0
MOVL C00324 V=800.0 PL=0
MOVL C00325 V=800.0 PL=0
MOVL C00326 V=800.0 PL=0
MOVL C00327 V=800.0 PL=0
MOVL C00328 V=800.0 PL=0
MOVL C00329 V=800.0 PL=0
MOVL C00330 V=800.0 PL=0
MOVL C00331 V=800.0 PL=0
MOVL C00332 V=800.0 PL=0
MOVL C00333 V=800.0 PL=0
MOVL C00334 V=800.0 PL=0
MOVL C00335 V=800.0 PL=0
MOVL C00336 V=800.0 PL=0
MOVL C00337 V=800.0 PL=0
MOVL C00338 V=800.0 PL=0
MOVL C00339 V=800.0 PL=0
MOVL C00340 V=800.0 PL=0
MOVL C00341 V=800.0 PL=0
MOVL C00342 V=800.0 PL=0
MOVL C00343 V=800.0 PL=0
MOVL C00344 V=800.0 PL=0
MOVL C00345 V=800.0 PL=0
MOVL C00346 V=800.0 PL=0
MOVL C00347 V=800.0 PL=0
MOVL C00348 V=800.0 PL=0
MOVL C00349 V=800.0 PL=0
MOVL C00350 V=800.0 PL=0
MOVL C00351 V=800.0 PL=0
MOVL C00352 V=800.0 PL=0
MOVL C00353 V=800.0 PL=0
MOVL C00354 V=800.0 PL=0
MOVL C00355 V=800.0 PL=0
MOVL C00356 V=800.0 PL=0
MOVL C00357 V=800.0 PL=0
MOVL C00358 V=800.0 PL=0
MOVL C00359 V=800.0 PL=0
MOVL C00360 V=800.0 PL=0
MOVL C00361 V=800.0 PL=0
MOVL C00362 V=800.0 PL=0
MOVL C00363 V=800.0 PL=0
MOVL C00364 V=800.0 PL=0
MOVL C00365 V=800.0 PL=0
MOVL C00366 V=800.0 PL=0
MOVL C00367 V=800.0 PL=0
MOVL C00368 V=800.0 PL=0
MOVL C00369 V=800.0 PL=0
MOVL C00370 V=800.0 PL=0
MOVL C00371 V=800.0 PL=0
MOVL C00372 V=800.0 PL=0
MOVL C00373 V=800.0 PL=0
MOVL C00374 V=800.0 PL=0
MOVL C00375 V=800.0 PL=0
MOVL C00376 V=800.0 PL=0
MOVL C00377 V=800.0 PL=0
MOVL C00378 V=800.0 PL=0
MOVL C00379 V=800.0 PL=0
MOVL C00380 V=800.0 PL=0
MOVL C00381 V=800.0 PL=0
MOVL C00382 V=800.0 PL=0
MOVL C00383 V=800.0 PL=0
MOVL C00384 V=800.0 PL=0
MOVL C00385 V=800.0 PL=0
MOVL C00386 V=800.0 PL=0
MOVL C00387 V=800.0 PL=0
MOVL C00388 V=800.0 PL=0
MOVL C00389 V=800.0 PL=0
MOVL C00390 V=800.0 PL=0
MOVL C00391 V=800.0 PL=0
MOVL C00392 V=800.0 PL=0
MOVL C00393 V=800.0 PL=0
MOVL C00394 V=800.0 PL=0
MOVL C00395 V=800.0 PL=0
MOVL C00396 V=800.0 PL=0
MOVL C00397 V=800.0 PL=0
MOVL C00398 V=800.0 PL=0
MOVL C00399 V=800.0 PL=0
MOVL C00400 V=800.0 PL=0
MOVL C00401 V=800.0 PL=0
MOVL C00402 V=800.0 PL=0
MOVL C00403 V=800.0 PL=0
MOVL C00404 V=800.0 PL=0
MOVL C00405 V=800.0 PL=0
MOVL C00406 V=800.0 PL=0
MOVL C00407 V=800.0 PL=0
MOVL C00408 V=800.0 PL=0
MOVL C00409 V=800.0 PL=0
MOVL C00410 V=800.0 PL=0
MOVL C00411 V=800.0 PL=0
MOVL C00412 V=800.0 PL=0
MOVL C00413 V=800.0 PL=0
MOVL C00414 V=800.0 PL=0
MOVL C00415 V=800.0 PL=0
MOVL C00416 V=800.0 PL=0
MOVL C00417 V=800.0 PL=0
MOVL C00418 V=800.0 PL=0
MOVL C00419 V=800.0 PL=0
MOVL C00420 V=800.0 PL=0
MOVL C00421 V=800.0 PL=0
MOVL C00422 V=800.0 PL=0
MOVL C00423 V=800.0 PL=0
MOVL C00424 V=800.0 PL=0
MOVL C00425 V=800.0 PL=0
MOVL C00426 V=800.0 PL=0
MOVL C00427 V=800.0 PL=0
MOVL C00428 V=800.0 PL=0
MOVL C00429 V=800.0 PL=0
MOVL C00430 V=800.0 PL=0
MOVL C00431 V=800.0 PL=0
MOVL C00432 V=800.0 PL=0
MOVL C00433 V=800.0 PL=0
MOVL C00434 V=800.0 PL=0
MOVL C00435 V=800.0 PL=0
MOVL C00436 V=800.0 PL=0
MOVL C00437 V=800.0 PL=0
MOVL C00438 V=800.0 PL=0
MOVL C00439 V=800.0 PL=0
MOVL C00440 V=800.0 PL=0
MOVL C00441 V=800.0 PL=0
MOVL C00442 V=800.0 PL=0
MOVL C00443 V=800.0 PL=0
MOVL C00444 V=800.0 PL=0
MOVL C00445 V=800.0 PL=0
MOVL C00446 V=800.0 PL=0
MOVL C00447 V=800.0 PL=0
MOVL C00448 V=800.0 PL=0
MOVL C00449 V=800.0 PL=0
MOVL C00450 V=800.0 PL=0
MOVL C00451 V=800.0 PL=0
MOVL C00452 V=800.0 PL=0
MOVL C00453 V=800.0 PL=0
MOVL C00454 V=800.0 PL=0
MOVL C00455 V=800.0 PL=0
MOVL C00456 V=800.0 PL=0
MOVL C00457 V=800.0 PL=0
MOVL C00458 V=800.0 PL=0
MOVL C00459 V=800.0 PL=0
MOVL C00460 V=800.0 PL=0
MOVL C00461 V=800.0 PL=0
MOVL C00462 V=800.0 PL=0
MOVL C00463 V=800.0 PL=0
MOVL C00464 V=800.0 PL=0
MOVL C00465 V=800.0 PL=0
MOVL C00466 V=800.0 PL=0
MOVL C00467 V=800.0 PL=0
MOVL C00468 V=800.0 PL=0
MOVL C00469 V=800.0 PL=0
MOVL C00470 V=800.0 PL=0
MOVL C00471 V=800.0 PL=0
MOVL C00472 V=800.0 PL=0
MOVL C00473 V=800.0 PL=0
MOVL C00474 V=800.0 PL=0
MOVL C00475 V=800.0 PL=0
MOVL C00476 V=800.0 PL=0
MOVL C00477 V=800.0 PL=0
MOVL C00478 V=800.0 PL=0
MOVL C00479 V=800.0 PL=0
MOVL C00480 V=800.0 PL=0
MOVL C00481 V=800.0 PL=0
MOVL C00482 V=800.0 PL=0
MOVL C00483 V=800.0 PL=0
MOVL C00484 V=800.0 PL=0
MOVL C00485 V=800.0 PL=0
MOVL C00486 V=800.0 PL=0
MOVL C00487 V=800.0 PL=0
MOVL C00488 V=800.0 PL=0
MOVL C00489 V=800.0 PL=0
MOVL C00490 V=800.0 PL=0
MOVL C00491 V=800.0 PL=0
MOVL C00492 V=800.0 PL=0
MOVL C00493 V=800.0 PL=0
MOVL C00494 V=800.0 PL=0
MOVL C00495 V=800.0 PL=0
MOVL C00496 V=800.0 PL=0
MOVL C00497 V=800.0 PL=0
MOVL C00498 V=800.0 PL=0
MOVL C00499 V=800.0 PL=0
MOVL C00500 V=800.0 PL=0
MOVL C00501 V=800.0 PL=0
MOVL C00502 V=800.0 PL=0
MOVL C00503 V=800.0 PL=0
MOVL C00504 V=800.0 PL=0
MOVL C00505 V=800.0 PL=0
MOVL C00506 V=800.0 PL=0
MOVL C00507 V=800.0 PL=0
MOVL C00508 V=800.0 PL=0
MOVL C00509 V=800.0 PL=0
MOVL C00510 V=800.0 PL=0
MOVL C00511 V=800.0 PL=0
MOVL C00512 V=800.0 PL=0
MOVL C00513 V=800.0 PL=0
MOVL C00514 V=800.0 PL=0
MOVL C00515 V=800.0 PL=0
MOVL C00516 V=800.0 PL=0
MOVL C00517 V=800.0 PL=0
MOVL C00518 V=800.0 PL=0
MOVL C00519 V=800.0 PL=0
MOVL C00520 V=800.0 PL=0
MOVL C00521 V=800.0 PL=0
MOVL C00522 V=800.0 PL=0
MOVL C00523 V=800.0 PL=0
MOVL C00524 V=800.0 PL=0
MOVL C00525 V=800.0 PL=0
MOVL C00526 V=800.0 PL=0
MOVL C00527 V=800.0 PL=0
MOVL C00528 V=800.0 PL=0
MOVL C00529 V=800.0 PL=0
MOVL C00530 V=800.0 PL=0
MOVL C00531 V=800.0 PL=0
MOVL C00532 V=800.0 PL=0
MOVL C00533 V=800.0 PL=0
MOVL C00534 V=800.0 PL=0
MOVL C00535 V=800.0 PL=0
MOVL C00536 V=800.0 PL=0
MOVL C00537 V=800.0 PL=0
MOVL C00538 V=800.0 PL=0
MOVL C00539 V=800.0 PL=0
MOVL C00540 V=800.0 PL=0
MOVL C00541 V=800.0 PL=0
MOVL C00542 V=800.0 PL=0
MOVL C00543 V=800.0 PL=0
MOVL C00544 V=800.0 PL=0
MOVL C00545 V=800.0 PL=0
MOVL C00546 V=800.0 PL=0
MOVL C00547 V=800.0 PL=0
MOVL C00548 V=800.0 PL=0
MOVL C00549 V=800.0 PL=0
MOVL C00550 V=800.0 PL=0
MOVL C00551 V=800.0 PL=0
MOVL C00552 V=800.0 PL=0
MOVL C00553 V=800.0 PL=0
MOVL C00554 V=800.0 PL=0
MOVL C00555 V=800.0 PL=0
MOVL C00556 V=800.0 PL=0
MOVL C00557 V=800.0 PL=0
MOVL C00558 V=800.0 PL=0
MOVL C00559 V=800.0 PL=0
MOVL C00560 V=800.0 PL=0
MOVL C00561 V=800.0 PL=0
MOVL C00562 V=800.0 PL=0
MOVL C00563 V=800.0 PL=0
MOVL C00564 V=800.0 PL=0
MOVL C00565 V=800.0 PL=0
MOVL C00566 V=800.0 PL=0
MOVL C00567 V=800.0 PL=0
MOVL C00568 V=800.0 PL=0
MOVL C00569 V=800.0 PL=0
MOVL C00570 V=800.0 PL=0
MOVL C00571 V=800.0 PL=0
MOVL C00572 V=800.0 PL=0
MOVL C00573 V=800.0 PL=0
MOVL C00574 V=800.0 PL=0
MOVL C00575 V=800.0 PL=0
MOVL C00576 V=800.0 PL=0
MOVL C00577 V=800.0 PL=0
MOVL C00578 V=800.0 PL=0
MOVL C00579 V=800.0 PL=0
MOVL C00580 V=800.0 PL=0
MOVL C00581 V=800.0 PL=0
MOVL C00582 V=800.0 PL=0
MOVL C00583 V=800.0 PL=0
MOVL C00584 V=800.0 PL=0
MOVL C00585 V=800.0 PL=0
MOVL C00586 V=800.0 PL=0
MOVL C00587 V=800.0 PL=0
MOVL C00588 V=800.0 PL=0
MOVL C00589 V=800.0 PL=0
MOVL C00590 V=800.0 PL=0
MOVL C00591 V=800.0 PL=0
MOVL C00592 V=800.0 PL=0
MOVL C00593 V=800.0 PL=0
MOVL C00594 V=800.0 PL=0
MOVL C00595 V=800.0 PL=0
MOVL C00596 V=800.0 PL=0
MOVL C00597 V=800.0 PL=0
MOVL C00598 V=800.0 PL=0
MOVL C00599 V=800.0 PL=0
MOVL C00600 V=800.0 PL=0
MOVL C00601 V=800.0 PL=0
MOVL C00602 V=800.0 PL=0
MOVL C00603 V=800.0 PL=0
MOVL C00604 V=800.0 PL=0
MOVL C00605 V=800.0 PL=0
MOVL C00606 V=800.0 PL=0
MOVL C00607 V=800.0 PL=0
MOVL C00608 V=800.0 PL=0
MOVL C00609 V=800.0 PL=0
MOVL C00610 V=800.0 PL=0
MOVL C00611 V=800.0 PL=0
MOVL C00612 V=800.0 PL=0
MOVL C00613 V=800.0 PL=0
MOVL C00614 V=800.0 PL=0
MOVL C00615 V=800.0 PL=0
MOVL C00616 V=800.0 PL=0
MOVL C00617 V=800.0 PL=0
MOVL C00618 V=800.0 PL=0
MOVL C00619 V=800.0 PL=0
MOVL C00620 V=800.0 PL=0
MOVL C00621 V=800.0 PL=0
MOVL C00622 V=800.0 PL=0
MOVL C00623 V=800.0 PL=0
MOVL C00624 V=800.0 PL=0
MOVL C00625 V=800.0 PL=0
MOVL C00626 V=800.0 PL=0
MOVL C00627 V=800.0 PL=0
MOVL C00628 V=800.0 PL=0
MOVL C00629 V=800.0 PL=0
MOVL C00630 V=800.0 PL=0
MOVL C00631 V=800.0 PL=0
MOVL C00632 V=800.0 PL=0
MOVL C00633 V=800.0 PL=0
MOVL C00634 V=800.0 PL=0
MOVL C00635 V=800.0 PL=0
MOVL C00636 V=800.0 PL=0
MOVL C00637 V=800.0 PL=0
MOVL C00638 V=800.0 PL=0
MOVL C00639 V=800.0 PL=0
MOVL C00640 V=800.0 PL=0
MOVL C00641 V=800.0 PL=0
MOVL C00642 V=800.0 PL=0
MOVL C00643 V=800.0 PL=0
MOVL C00644 V=800.0 PL=0
MOVL C00645 V=800.0 PL=0
MOVL C00646 V=800.0 PL=0
MOVL C00647 V=800.0 PL=0
MOVL C00648 V=800.0 PL=0
MOVL C00649 V=800.0 PL=0
MOVL C00650 V=800.0 PL=0
MOVL C00651 V=800.0 PL=0
MOVL C00652 V=800.0 PL=0
MOVL C00653 V=800.0 PL=0
MOVL C00654 V=800.0 PL=0
MOVL C00655 V=800.0 PL=0
MOVL C00656 V=800.0 PL=0
MOVL C00657 V=800.0 PL=0
MOVL C00658 V=800.0 PL=0
MOVL C00659 V=800.0 PL=0
MOVL C00660 V=800.0 PL=0
MOVL C00661 V=800.0 PL=0
MOVL C00662 V=800.0 PL=0
MOVL C00663 V=800.0 PL=0
MOVL C00664 V=800.0 PL=0
MOVL C00665 V=800.0 PL=0
MOVL C00666 V=800.0 PL=0
MOVL C00667 V=800.0 PL=0
MOVL C00668 V=800.0 PL=0
MOVL C00669 V=800.0 PL=0
MOVL C00670 V=800.0 PL=0
MOVL C00671 V=800.0 PL=0
MOVL C00672 V=800.0 PL=0
MOVL C00673 V=800.0 PL=0
MOVL C00674 V=800.0 PL=0
MOVL C00675 V=800.0 PL=0
MOVL C00676 V=800.0 PL=0
MOVL C00677 V=800.0 PL=0
MOVL C00678 V=800.0 PL=0
MOVL C00679 V=800.0 PL=0
MOVL C00680 V=800.0 PL=0
MOVL C00681 V=800.0 PL=0
MOVL C00682 V=800.0 PL=0
MOVL C00683 V=800.0 PL=0
MOVL C00684 V=800.0 PL=0
MOVL C00685 V=800.0 PL=0
MOVL C00686 V=800.0 PL=0
MOVL C00687 V=800.0 PL=0
MOVL C00688 V=800.0 PL=0
MOVL C00689 V=800.0 PL=0
MOVL C00690 V=800.0 PL=0
MOVL C00691 V=800.0 PL=0
MOVL C00692 V=800.0 PL=0
MOVL C00693 V=800.0 PL=0
MOVL C00694 V=800.0 PL=0
MOVL C00695 V=800.0 PL=0
MOVL C00696 V=800.0 PL=0
MOVL C00697 V=800.0 PL=0
MOVL C00698 V=800.0 PL=0
MOVL C00699 V=800.0 PL=0
MOVL C00700 V=800.0 PL=0
MOVL C00701 V=800.0 PL=0
MOVL C00702 V=800.0 PL=0
MOVL C00703 V=800.0 PL=0
MOVL C00704 V=800.0 PL=0
MOVL C00705 V=800.0 PL=0
MOVL C00706 V=800.0 PL=0
MOVL C00707 V=800.0 PL=0
MOVL C00708 V=800.0 PL=0
MOVL C00709 V=800.0 PL=0
MOVL C00710 V=800.0 PL=0
MOVL C00711 V=800.0 PL=0
MOVL C00712 V=800.0 PL=0
MOVL C00713 V=800.0 PL=0
MOVL C00714 V=800.0 PL=0
MOVL C00715 V=800.0 PL=0
MOVL C00716 V=800.0 PL=0
MOVL C00717 V=800.0 PL=0
MOVL C00718 V=800.0 PL=0
MOVL C00719 V=800.0 PL=0
MOVL C00720 V=800.0 PL=0
MOVL C00721 V=800.0 PL=0
MOVL C00722 V=800.0 PL=0
MOVL C00723 V=800.0 PL=0
MOVL C00724 V=800.0 PL=0
MOVL C00725 V=800.0 PL=0
MOVL C00726 V=800.0 PL=0
MOVL C00727 V=800.0 PL=0
MOVL C00728 V=800.0 PL=0
MOVL C00729 V=800.0 PL=0
MOVL C00730 V=800.0 PL=0
MOVL C00731 V=800.0 PL=0
MOVL C00732 V=800.0 PL=0
MOVL C00733 V=800.0 PL=0
MOVL C00734 V=800.0 PL=0
MOVL C00735 V=800.0 PL=0
MOVL C00736 V=800.0 PL=0
MOVL C00737 V=800.0 PL=0
MOVL C00738 V=800.0 PL=0
MOVL C00739 V=800.0 PL=0
MOVL C00740 V=800.0 PL=0
MOVL C00741 V=800.0 PL=0
MOVL C00742 V=800.0 PL=0
MOVL C00743 V=800.0 PL=0
MOVL C00744 V=800.0 PL=0
MOVL C00745 V=800.0 PL=0
MOVL C00746 V=800.0 PL=0
MOVL C00747 V=800.0 PL=0
MOVL C00748 V=800.0 PL=0
MOVL C00749 V=800.0 PL=0
MOVL C00750 V=800.0 PL=0
MOVL C00751 V=800.0 PL=0
MOVL C00752 V=800.0 PL=0
MOVL C00753 V=800.0 PL=0
MOVL C00754 V=800.0 PL=0
MOVL C00755 V=800.0 PL=0
MOVL C00756 V=800.0 PL=0
MOVL C00757 V=800.0 PL=0
MOVL C00758 V=800.0 PL=0
MOVL C00759 V=800.0 PL=0
MOVL C00760 V=800.0 PL=0
MOVL C00761 V=800.0 PL=0
MOVL C00762 V=800.0 PL=0
MOVL C00763 V=800.0 PL=0
MOVL C00764 V=800.0 PL=0
MOVL C00765 V=800.0 PL=0
MOVL C00766 V=800.0 PL=0
MOVL C00767 V=800.0 PL=0
MOVL C00768 V=800.0 PL=0
MOVL C00769 V=800.0 PL=0
MOVL C00770 V=800.0 PL=0
MOVL C00771 V=800.0 PL=0
MOVL C00772 V=800.0 PL=0
MOVL C00773 V=800.0 PL=0
MOVL C00774 V=800.0 PL=0
MOVL C00775 V=800.0 PL=0
MOVL C00776 V=800.0 PL=0
MOVL C00777 V=800.0 PL=0
MOVL C00778 V=800.0 PL=0
MOVL C00779 V=800.0 PL=0
MOVL C00780 V=800.0 PL=0
MOVL C00781 V=800.0 PL=0
MOVL C00782 V=800.0 PL=0
MOVL C00783 V=800.0 PL=0
MOVL C00784 V=800.0 PL=0
MOVL C00785 V=800.0 PL=0
MOVL C00786 V=800.0 PL=0
MOVL C00787 V=800.0 PL=0
MOVL C00788 V=800.0 PL=0
MOVL C00789 V=800.0 PL=0
MOVL C00790 V=800.0 PL=0
MOVL C00791 V=800.0 PL=0
MOVL C00792 V=800.0 PL=0
MOVL C00793 V=800.0 PL=0
MOVL C00794 V=800.0 PL=0
MOVL C00795 V=800.0 PL=0
MOVL C00796 V=800.0 PL=0
MOVL C00797 V=800.0 PL=0
MOVL C00798 V=800.0 PL=0
MOVL C00799 V=800.0 PL=0
MOVL C00800 V=800.0 PL=0
MOVL C00801 V=800.0 PL=0
MOVL C00802 V=800.0 PL=0
MOVL C00803 V=800.0 PL=0
MOVL C00804 V=800.0 PL=0
MOVL C00805 V=800.0 PL=0
MOVL C00806 V=800.0 PL=0
MOVL C00807 V=800.0 PL=0
MOVL C00808 V=800.0 PL=0
MOVL C00809 V=800.0 PL=0
MOVL C00810 V=800.0 PL=0
MOVL C00811 V=800.0 PL=0
MOVL C00812 V=800.0 PL=0
MOVL C00813 V=800.0 PL=0
MOVL C00814 V=800.0 PL=0
MOVL C00815 V=800.0 PL=0
MOVL C00816 V=800.0 PL=0
MOVL C00817 V=800.0 PL=0
MOVL C00818 V=800.0 PL=0
MOVL C00819 V=800.0 PL=0
MOVL C00820 V=800.0 PL=0
MOVL C00821 V=800.0 PL=0
MOVL C00822 V=800.0 PL=0
MOVL C00823 V=800.0 PL=0
MOVL C00824 V=800.0 PL=0
MOVL C00825 V=800.0 PL=0
MOVL C00826 V=800.0 PL=0
MOVL C00827 V=800.0 PL=0
MOVL C00828 V=800.0 PL=0
MOVL C00829 V=800.0 PL=0
MOVL C00830 V=800.0 PL=0
MOVL C00831 V=800.0 PL=0
MOVL C00832 V=800.0 PL=0
MOVL C00833 V=800.0 PL=0
MOVL C00834 V=800.0 PL=0
MOVL C00835 V=800.0 PL=0
MOVL C00836 V=800.0 PL=0
MOVL C00837 V=800.0 PL=0
MOVL C00838 V=800.0 PL=0
MOVL C00839 V=800.0 PL=0
MOVL C00840 V=800.0 PL=0
MOVL C00841 V=800.0 PL=0
MOVL C00842 V=800.0 PL=0
MOVL C00843 V=800.0 PL=0
MOVL C00844 V=800.0 PL=0
MOVL C00845 V=800.0 PL=0
MOVL C00846 V=800.0 PL=0
MOVL C00847 V=800.0 PL=0
MOVL C00848 V=800.0 PL=0
MOVL C00849 V=800.0 PL=0
MOVL C00850 V=800.0 PL=0
MOVL C00851 V=800.0 PL=0
MOVL C00852 V=800.0 PL=0
MOVL C00853 V=800.0 PL=0
MOVL C00854 V=800.0 PL=0
MOVL C00855 V=800.0 PL=0
MOVL C00856 V=800.0 PL=0
MOVL C00857 V=800.0 PL=0
MOVL C00858 V=800.0 PL=0
MOVL C00859 V=800.0 PL=0
MOVL C00860 V=800.0 PL=0
MOVL C00861 V=800.0 PL=0
MOVL C00862 V=800.0 PL=0
MOVL C00863 V=800.0 PL=0
MOVL C00864 V=800.0 PL=0
MOVL C00865 V=800.0 PL=0
MOVL C00866 V=800.0 PL=0
MOVL C00867 V=800.0 PL=0
MOVL C00868 V=800.0 PL=0
MOVL C00869 V=800.0 PL=0
MOVL C00870 V=800.0 PL=0
MOVL C00871 V=800.0 PL=0
MOVL C00872 V=800.0 PL=0
MOVL C00873 V=800.0 PL=0
MOVL C00874 V=800.0 PL=0
MOVL C00875 V=800.0 PL=0
MOVL C00876 V=800.0 PL=0
MOVL C00877 V=800.0 PL=0
MOVL C00878 V=800.0 PL=0
MOVL C00879 V=800.0 PL=0
MOVL C00880 V=800.0 PL=0
MOVL C00881 V=800.0 PL=0
MOVL C00882 V=800.0 PL=0
MOVL C00883 V=800.0 PL=0
MOVL C00884 V=800.0 PL=0
MOVL C00885 V=800.0 PL=0
MOVL C00886 V=800.0 PL=0
MOVL C00887 V=800.0 PL=0
MOVL C00888 V=800.0 PL=0
MOVL C00889 V=800.0 PL=0
MOVL C00890 V=800.0 PL=0
MOVL C00891 V=800.0 PL=0
MOVL C00892 V=800.0 PL=0
MOVL C00893 V=800.0 PL=0
MOVL C00894 V=800.0 PL=0
MOVL C00895 V=800.0 PL=0
MOVL C00896 V=800.0 PL=0
MOVL C00897 V=800.0 PL=0
MOVL C00898 V=800.0 PL=0
MOVL C00899 V=800.0 PL=0
MOVL C00900 V=800.0 PL=0
MOVL C00901 V=800.0 PL=0
MOVL C00902 V=800.0 PL=0
MOVL C00903 V=800.0 PL=0
MOVL C00904 V=800.0 PL=0
MOVL C00905 V=800.0 PL=0
MOVL C00906 V=800.0 PL=0
MOVL C00907 V=800.0 PL=0
MOVL C00908 V=800.0 PL=0
MOVL C00909 V=800.0 PL=0
MOVL C00910 V=800.0 PL=0
MOVL C00911 V=800.0 PL=0
MOVL C00912 V=800.0 PL=0
MOVL C00913 V=800.0 PL=0
MOVL C00914 V=800.0 PL=0
MOVL C00915 V=800.0 PL=0
MOVL C00916 V=800.0 PL=0
MOVL C00917 V=800.0 PL=0
MOVL C00918 V=800.0 PL=0
MOVL C00919 V=800.0 PL=0
MOVL C00920 V=800.0 PL=0
MOVL C00921 V=800.0 PL=0
MOVL C00922 V=800.0 PL=0
MOVL C00923 V=800.0 PL=0
MOVL C00924 V=800.0 PL=0
MOVL C00925 V=800.0 PL=0
MOVL C00926 V=800.0 PL=0
MOVL C00927 V=800.0 PL=0
MOVL C00928 V=800.0 PL=0
MOVL C00929 V=800.0 PL=0
MOVL C00930 V=800.0 PL=0
MOVL C00931 V=800.0 PL=0
MOVL C00932 V=800.0 PL=0
MOVL C00933 V=800.0 PL=0
MOVL C00934 V=800.0 PL=0
MOVL C00935 V=800.0 PL=0
MOVL C00936 V=800.0 PL=0
MOVL C00937 V=800.0 PL=0
MOVL C00938 V=800.0 PL=0
MOVL C00939 V=800.0 PL=0
MOVL C00940 V=800.0 PL=0
MOVL C00941 V=800.0 PL=0
MOVL C00942 V=800.0 PL=0
MOVL C00943 V=800.0 PL=0
MOVL C00944 V=800.0 PL=0
MOVL C00945 V=800.0 PL=0
MOVL C00946 V=800.0 PL=0
MOVL C00947 V=800.0 PL=0
MOVL C00948 V=800.0 PL=0
MOVL C00949 V=800.0 PL=0
MOVL C00950 V=800.0 PL=0
MOVL C00951 V=800.0 PL=0
MOVL C00952 V=800.0 PL=0
MOVL C00953 V=800.0 PL=0
MOVL C00954 V=800.0 PL=0
MOVL C00955 V=800.0 PL=0
MOVL C00956 V=800.0 PL=0
MOVL C00957 V=800.0 PL=0
MOVL C00958 V=800.0 PL=0
MOVL C00959 V=800.0 PL=0
MOVL C00960 V=800.0 PL=0
MOVL C00961 V=800.0 PL=0
MOVL C00962 V=800.0 PL=0
MOVL C00963 V=800.0 PL=0
MOVL C00964 V=800.0 PL=0
MOVL C00965 V=800.0 PL=0
MOVL C00966 V=800.0 PL=0
MOVL C00967 V=800.0 PL=0
MOVL C00968 V=800.0 PL=0
MOVL C00969 V=800.0 PL=0
MOVL C00970 V=800.0 PL=0
MOVL C00971 V=800.0 PL=0
MOVL C00972 V=800.0 PL=0
MOVL C00973 V=800.0 PL=0
MOVL C00974 V=800.0 PL=0
MOVL C00975 V=800.0 PL=0
MOVL C00976 V=800.0 PL=0
MOVL C00977 V=800.0 PL=0
MOVL C00978 V=800.0 PL=0
MOVL C00979 V=800.0 PL=0
MOVL C00980 V=800.0 PL=0
MOVL C00981 V=800.0 PL=0
MOVL C00982 V=800.0 PL=0
MOVL C00983 V=800.0 PL=0
MOVL C00984 V=800.0 PL=0
MOVL C00985 V=800.0 PL=0
MOVL C00986 V=800.0 PL=0
MOVL C00987 V=800.0 PL=0
MOVL C00988 V=800.0 PL=0
MOVL C00989 V=800.0 PL=0
MOVL C00990 V=800.0 PL=0
MOVL C00991 V=800.0 PL=0
MOVL C00992 V=800.0 PL=0
MOVL C00993 V=800.0 PL=0
MOVL C00994 V=800.0 PL=0
MOVL C00995 V=800.0 PL=0
MOVL C00996 V=800.0 PL=0
MOVL C00997 V=800.0 PL=0
MOVL C00998 V=800.0 PL=0
MOVL C00999 V=800.0 PL=0
MOVL C01000 V=800.0 PL=0
MOVL C01001 V=800.0 PL=0
MOVL C01002 V=800.0 PL=0
MOVL C01003 V=800.0 PL=0
MOVL C01004 V=800.0 PL=0
MOVL C01005 V=800.0 PL=0
MOVL C01006 V=800.0 PL=0
MOVL C01007 V=800.0 PL=0
MOVL C01008 V=800.0 PL=0
MOVL C01009 V=800.0 PL=0
MOVL C01010 V=800.0 PL=0
MOVL C01011 V=800.0 PL=0
MOVL C01012 V=800.0 PL=0
MOVL C01013 V=800.0 PL=0
MOVL C01014 V=800.0 PL=0
MOVL C01015 V=800.0 PL=0
MOVL C01016 V=800.0 PL=0
MOVL C01017 V=800.0 PL=0
MOVL C01018 V=800.0 PL=0
MOVL C01019 V=800.0 PL=0
MOVL C01020 V=800.0 PL=0
MOVL C01021 V=800.0 PL=0
MOVL C01022 V=800.0 PL=0
MOVL C01023 V=800.0 PL=0
MOVL C01024 V=800.0 PL=0
MOVL C01025 V=800.0 PL=0
MOVL C01026 V=800.0 PL=0
MOVL C01027 V=800.0 PL=0
MOVL C01028 V=800.0 PL=0
MOVL C01029 V=800.0 PL=0
MOVL C01030 V=800.0 PL=0
MOVL C01031 V=800.0 PL=0
MOVL C01032 V=800.0 PL=0
MOVL C01033 V=800.0 PL=0
MOVL C01034 V=800.0 PL=0
MOVL C01035 V=800.0 PL=0
MOVL C01036 V=800.0 PL=0
MOVL C01037 V=800.0 PL=0
MOVL C01038 V=800.0 PL=0
MOVL C01039 V=800.0 PL=0
MOVL C01040 V=800.0 PL=0
MOVL C01041 V=800.0 PL=0
MOVL C01042 V=800.0 PL=0
MOVL C01043 V=800.0 PL=0
MOVL C01044 V=800.0 PL=0
MOVL C01045 V=800.0 PL=0
MOVL C01046 V=800.0 PL=0
MOVL C01047 V=800.0 PL=0
MOVL C01048 V=800.0 PL=0
MOVL C01049 V=800.0 PL=0
MOVL C01050 V=800.0 PL=0
MOVL C01051 V=800.0 PL=0
MOVL C01052 V=800.0 PL=0
MOVL C01053 V=800.0 PL=0
MOVL C01054 V=800.0 PL=0
MOVL C01055 V=800.0 PL=0
MOVL C01056 V=800.0 PL=0
MOVL C01057 V=800.0 PL=0
MOVL C01058 V=800.0 PL=0
MOVL C01059 V=800.0 PL=0
MOVL C01060 V=800.0 PL=0
MOVL C01061 V=800.0 PL=0
MOVL C01062 V=800.0 PL=0
MOVL C01063 V=800.0 PL=0
MOVL C01064 V=800.0 PL=0
MOVL C01065 V=800.0 PL=0
MOVL C01066 V=800.0 PL=0
MOVL C01067 V=800.0 PL=0
MOVL C01068 V=800.0 PL=0
MOVL C01069 V=800.0 PL=0
MOVL C01070 V=800.0 PL=0
MOVL C01071 V=800.0 PL=0
MOVL C01072 V=800.0 PL=0
MOVL C01073 V=800.0 PL=0
MOVL C01074 V=800.0 PL=0
MOVL C01075 V=800.0 PL=0
MOVL C01076 V=800.0 PL=0
MOVL C01077 V=800.0 PL=0
MOVL C01078 V=800.0 PL=0
MOVL C01079 V=800.0 PL=0
MOVL C01080 V=800.0 PL=0
MOVL C01081 V=800.0 PL=0
MOVL C01082 V=800.0 PL=0
MOVL C01083 V=800.0 PL=0
MOVL C01084 V=800.0 PL=0
MOVL C01085 V=800.0 PL=0
MOVL C01086 V=800.0 PL=0
MOVL C01087 V=800.0 PL=0
MOVL C01088 V=800.0 PL=0
MOVL C01089 V=800.0 PL=0
MOVL C01090 V=800.0 PL=0
MOVL C01091 V=800.0 PL=0
MOVL C01092 V=800.0 PL=0
MOVL C01093 V=800.0 PL=0
MOVL C01094 V=800.0 PL=0
MOVL C01095 V=800.0 PL=0
MOVL C01096 V=800.0 PL=0
MOVL C01097 V=800.0 PL=0
MOVL C01098 V=800.0 PL=0
MOVL C01099 V=800.0 PL=0
MOVL C01100 V=800.0 PL=0
MOVL C01101 V=800.0 PL=0
MOVL C01102 V=800.0 PL=0
MOVL C01103 V=800.0 PL=0
MOVL C01104 V=800.0 PL=0
MOVL C01105 V=800.0 PL=0
MOVL C01106 V=800.0 PL=0
MOVL C01107 V=800.0 PL=0
MOVL C01108 V=800.0 PL=0
MOVL C01109 V=800.0 PL=0
MOVL C01110 V=800.0 PL=0
MOVL C01111 V=800.0 PL=0
MOVL C01112 V=800.0 PL=0
MOVL C01113 V=800.0 PL=0
MOVL C01114 V=800.0 PL=0
MOVL C01115 V=800.0 PL=0
MOVL C01116 V=800.0 PL=0
MOVL C01117 V=800.0 PL=0
MOVL C01118 V=800.0 PL=0
MOVL C01119 V=800.0 PL=0
MOVL C01120 V=800.0 PL=0
MOVL C01121 V=800.0 PL=0
MOVL C01122 V=800.0 PL=0
MOVL C01123 V=800.0 PL=0
MOVL C01124 V=800.0 PL=0
MOVL C01125 V=800.0 PL=0
MOVL C01126 V=800.0 PL=0
MOVL C01127 V=800.0 PL=0
MOVL C01128 V=800.0 PL=0
MOVL C01129 V=800.0 PL=0
MOVL C01130 V=800.0 PL=0
MOVL C01131 V=800.0 PL=0
MOVL C01132 V=800.0 PL=0
MOVL C01133 V=800.0 PL=0
MOVL C01134 V=800.0 PL=0
MOVL C01135 V=800.0 PL=0
MOVL C01136 V=800.0 PL=0
MOVL C01137 V=800.0 PL=0
MOVL C01138 V=800.0 PL=0
MOVL C01139 V=800.0 PL=0
MOVL C01140 V=800.0 PL=0
MOVL C01141 V=800.0 PL=0
MOVL C01142 V=800.0 PL=0
MOVL C01143 V=800.0 PL=0
MOVL C01144 V=800.0 PL=0
MOVL C01145 V=800.0 PL=0
MOVL C01146 V=800.0 PL=0
MOVL C01147 V=800.0 PL=0
MOVL C01148 V=800.0 PL=0
MOVL C01149 V=800.0 PL=0
MOVL C01150 V=800.0 PL=0
MOVL C01151 V=800.0 PL=0
MOVL C01152 V=800.0 PL=0
MOVL C01153 V=800.0 PL=0
MOVL C01154 V=800.0 PL=0
MOVL C01155 V=800.0 PL=0
MOVL C01156 V=800.0 PL=0
MOVL C01157 V=800.0 PL=0
MOVL C01158 V=800.0 PL=0
MOVL C01159 V=800.0 PL=0
MOVL C01160 V=800.0 PL=0
MOVL C01161 V=800.0 PL=0
MOVL C01162 V=800.0 PL=0
MOVL C01163 V=800.0 PL=0
MOVL C01164 V=800.0 PL=0
MOVL C01165 V=800.0 PL=0
MOVL C01166 V=800.0 PL=0
MOVL C01167 V=800.0 PL=0
MOVL C01168 V=800.0 PL=0
MOVL C01169 V=800.0 PL=0
MOVL C01170 V=800.0 PL=0
MOVL C01171 V=800.0 PL=0
MOVL C01172 V=800.0 PL=0
MOVL C01173 V=800.0 PL=0
MOVL C01174 V=800.0 PL=0
MOVL C01175 V=800.0 PL=0
MOVL C01176 V=800.0 PL=0
MOVL C01177 V=800.0 PL=0
MOVL C01178 V=800.0 PL=0
MOVL C01179 V=800.0 PL=0
MOVL C01180 V=800.0 PL=0
MOVL C01181 V=800.0 PL=0
MOVL C01182 V=800.0 PL=0
MOVL C01183 V=800.0 PL=0
MOVL C01184 V=800.0 PL=0
MOVL C01185 V=800.0 PL=0
MOVL C01186 V=800.0 PL=0
MOVL C01187 V=800.0 PL=0
MOVL C01188 V=800.0 PL=0
MOVL C01189 V=800.0 PL=0
MOVL C01190 V=800.0 PL=0
MOVL C01191 V=800.0 PL=0
MOVL C01192 V=800.0 PL=0
MOVL C01193 V=800.0 PL=0
MOVL C01194 V=800.0 PL=0
MOVL C01195 V=800.0 PL=0
MOVL C01196 V=800.0 PL=0
MOVL C01197 V=800.0 PL=0
MOVL C01198 V=800.0 PL=0
MOVL C01199 V=800.0 PL=0
MOVL C01200 V=800.0 PL=0
MOVL C01201 V=800.0 PL=0
MOVL C01202 V=800.0 PL=0
MOVL C01203 V=800.0 PL=0
MOVL C01204 V=800.0 PL=0
MOVL C01205 V=800.0 PL=0
MOVL C01206 V=800.0 PL=0
MOVL C01207 V=800.0 PL=0
MOVL C01208 V=800.0 PL=0
MOVL C01209 V=800.0 PL=0
MOVL C01210 V=800.0 PL=0
MOVL C01211 V=800.0 PL=0
MOVL C01212 V=800.0 PL=0
MOVL C01213 V=800.0 PL=0
MOVL C01214 V=800.0 PL=0
MOVL C01215 V=800.0 PL=0
MOVL C01216 V=800.0 PL=0
MOVL C01217 V=800.0 PL=0
MOVL C01218 V=800.0 PL=0
MOVL C01219 V=800.0 PL=0
MOVL C01220 V=800.0 PL=0
MOVL C01221 V=800.0 PL=0
MOVL C01222 V=800.0 PL=0
MOVL C01223 V=800.0 PL=0
MOVL C01224 V=800.0 PL=0
MOVL C01225 V=800.0 PL=0
MOVL C01226 V=800.0 PL=0
MOVL C01227 V=800.0 PL=0
MOVL C01228 V=800.0 PL=0
MOVL C01229 V=800.0 PL=0
MOVL C01230 V=800.0 PL=0
MOVL C01231 V=800.0 PL=0
MOVL C01232 V=800.0 PL=0
MOVL C01233 V=800.0 PL=0
MOVL C01234 V=800.0 PL=0
MOVL C01235 V=800.0 PL=0
MOVL C01236 V=800.0 PL=0
MOVL C01237 V=800.0 PL=0
MOVL C01238 V=800.0 PL=0
MOVL C01239 V=800.0 PL=0
MOVL C01240 V=800.0 PL=0
MOVL C01241 V=800.0 PL=0
MOVL C01242 V=800.0 PL=0
MOVL C01243 V=800.0 PL=0
MOVL C01244 V=800.0 PL=0
MOVL C01245 V=800.0 PL=0
MOVL C01246 V=800.0 PL=0
MOVL C01247 V=800.0 PL=0
MOVL C01248 V=800.0 PL=0
MOVL C01249 V=800.0 PL=0
MOVL C01250 V=800.0 PL=0
MOVL C01251 V=800.0 PL=0
MOVL C01252 V=800.0 PL=0
MOVL C01253 V=800.0 PL=0
MOVL C01254 V=800.0 PL=0
MOVL C01255 V=800.0 PL=0
MOVL C01256 V=800.0 PL=0
MOVL C01257 V=800.0 PL=0
MOVL C01258 V=800.0 PL=0
MOVL C01259 V=800.0 PL=0
MOVL C01260 V=800.0 PL=0
MOVL C01261 V=800.0 PL=0
MOVL C01262 V=800.0 PL=0
MOVL C01263 V=800.0 PL=0
MOVL C01264 V=800.0 PL=0
MOVL C01265 V=800.0 PL=0
MOVL C01266 V=800.0 PL=0
MOVL C01267 V=800.0 PL=0
MOVL C01268 V=800.0 PL=0
MOVL C01269 V=800.0 PL=0
MOVL C01270 V=800.0 PL=0
MOVL C01271 V=800.0 PL=0
MOVL C01272 V=800.0 PL=0
MOVL C01273 V=800.0 PL=0
MOVL C01274 V=800.0 PL=0
MOVL C01275 V=800.0 PL=0
MOVL C01276 V=800.0 PL=0
MOVL C01277 V=800.0 PL=0
MOVL C01278 V=800.0 PL=0
MOVL C01279 V=800.0 PL=0
MOVL C01280 V=800.0 PL=0
MOVL C01281 V=800.0 PL=0
MOVL C01282 V=800.0 PL=0
MOVL C01283 V=800.0 PL=0
MOVL C01284 V=800.0 PL=0
MOVL C01285 V=800.0 PL=0
MOVL C01286 V=800.0 PL=0
MOVL C01287 V=800.0 PL=0
MOVL C01288 V=800.0 PL=0
MOVL C01289 V=800.0 PL=0
MOVL C01290 V=800.0 PL=0
MOVL C01291 V=800.0 PL=0
MOVL C01292 V=800.0 PL=0
MOVL C01293 V=800.0 PL=0
MOVL C01294 V=800.0 PL=0
MOVL C01295 V=800.0 PL=0
MOVL C01296 V=800.0 PL=0
MOVL C01297 V=800.0 PL=0
MOVL C01298 V=800.0 PL=0
MOVL C01299 V=800.0 PL=0
MOVL C01300 V=800.0 PL=0
MOVL C01301 V=800.0 PL=0
MOVL C01302 V=800.0 PL=0
MOVL C01303 V=800.0 PL=0
MOVL C01304 V=800.0 PL=0
MOVL C01305 V=800.0 PL=0
MOVL C01306 V=800.0 PL=0
MOVL C01307 V=800.0 PL=0
MOVL C01308 V=800.0 PL=0
MOVL C01309 V=800.0 PL=0
MOVL C01310 V=800.0 PL=0
MOVL C01311 V=800.0 PL=0
MOVL C01312 V=800.0 PL=0
MOVL C01313 V=800.0 PL=0
MOVL C01314 V=800.0 PL=0
MOVL C01315 V=800.0 PL=0
MOVL C01316 V=800.0 PL=0
MOVL C01317 V=800.0 PL=0
MOVL C01318 V=800.0 PL=0
MOVL C01319 V=800.0 PL=0
MOVL C01320 V=800.0 PL=0
MOVL C01321 V=800.0 PL=0
MOVL C01322 V=800.0 PL=0
MOVL C01323 V=800.0 PL=0
MOVL C01324 V=800.0 PL=0
MOVL C01325 V=800.0 PL=0
MOVL C01326 V=800.0 PL=0
MOVL C01327 V=800.0 PL=0
MOVL C01328 V=800.0 PL=0
MOVL C01329 V=800.0 PL=0
MOVL C01330 V=800.0 PL=0
MOVL C01331 V=800.0 PL=0
MOVL C01332 V=800.0 PL=0
MOVL C01333 V=800.0 PL=0
MOVL C01334 V=800.0 PL=0
MOVL C01335 V=800.0 PL=0
MOVL C01336 V=800.0 PL=0
MOVL C01337 V=800.0 PL=0
MOVL C01338 V=800.0 PL=0
MOVL C01339 V=800.0 PL=0
MOVL C01340 V=800.0 PL=0
MOVL C01341 V=800.0 PL=0
MOVL C01342 V=800.0 PL=0
MOVL C01343 V=800.0 PL=0
MOVL C01344 V=800.0 PL=0
MOVL C01345 V=800.0 PL=0
MOVL C01346 V=800.0 PL=0
MOVL C01347 V=800.0 PL=0
MOVL C01348 V=800.0 PL=0
MOVL C01349 V=800.0 PL=0
MOVL C01350 V=800.0 PL=0
MOVL C01351 V=800.0 PL=0
MOVL C01352 V=800.0 PL=0
MOVL C01353 V=800.0 PL=0
MOVL C01354 V=800.0 PL=0
MOVL C01355 V=800.0 PL=0
MOVL C01356 V=800.0 PL=0
MOVL C01357 V=800.0 PL=0
MOVL C01358 V=800.0 PL=0
MOVL C01359 V=800.0 PL=0
MOVL C01360 V=800.0 PL=0
MOVL C01361 V=800.0 PL=0
MOVL C01362 V=800.0 PL=0
MOVL C01363 V=800.0 PL=0
MOVL C01364 V=800.0 PL=0
MOVL C01365 V=800.0 PL=0
MOVL C01366 V=800.0 PL=0
MOVL C01367 V=800.0 PL=0
MOVL C01368 V=800.0 PL=0
MOVL C01369 V=800.0 PL=0
MOVL C01370 V=800.0 PL=0
MOVL C01371 V=800.0 PL=0
MOVL C01372 V=800.0 PL=0
MOVL C01373 V=800.0 PL=0
MOVL C01374 V=800.0 PL=0
MOVL C01375 V=800.0 PL=0
MOVL C01376 V=800.0 PL=0
MOVL C01377 V=800.0 PL=0
MOVL C01378 V=800.0 PL=0
MOVL C01379 V=800.0 PL=0
MOVL C01380 V=800.0 PL=0
MOVL C01381 V=800.0 PL=0
MOVL C01382 V=800.0 PL=0
MOVL C01383 V=800.0 PL=0
MOVL C01384 V=800.0 PL=0
MOVL C01385 V=800.0 PL=0
MOVL C01386 V=800.0 PL=0
MOVL C01387 V=800.0 PL=0
MOVL C01388 V=800.0 PL=0
MOVL C01389 V=800.0 PL=0
MOVL C01390 V=800.0 PL=0
MOVL C01391 V=800.0 PL=0
MOVL C01392 V=800.0 PL=0
MOVL C01393 V=800.0 PL=0
MOVL C01394 V=800.0 PL=0
MOVL C01395 V=800.0 PL=0
MOVL C01396 V=800.0 PL=0
MOVL C01397 V=800.0 PL=0
MOVL C01398 V=800.0 PL=0
MOVL C01399 V=800.0 PL=0
MOVL C01400 V=800.0 PL=0
MOVL C01401 V=800.0 PL=0
MOVL C01402 V=800.0 PL=0
MOVL C01403 V=800.0 PL=0
MOVL C01404 V=800.0 PL=0
MOVL C01405 V=800.0 PL=0
MOVL C01406 V=800.0 PL=0
MOVL C01407 V=800.0 PL=0
MOVL C01408 V=800.0 PL=0
MOVL C01409 V=800.0 PL=0
MOVL C01410 V=800.0 PL=0
MOVL C01411 V=800.0 PL=0
MOVL C01412 V=800.0 PL=0
MOVL C01413 V=800.0 PL=0
MOVL C01414 V=800.0 PL=0
MOVL C01415 V=800.0 PL=0
MOVL C01416 V=800.0 PL=0
MOVL C01417 V=800.0 PL=0
MOVL C01418 V=800.0 PL=0
MOVL C01419 V=800.0 PL=0
MOVL C01420 V=800.0 PL=0
MOVL C01421 V=800.0 PL=0
MOVL C01422 V=800.0 PL=0
MOVL C01423 V=800.0 PL=0
MOVL C01424 V=800.0 PL=0
MOVL C01425 V=800.0 PL=0
MOVL C01426 V=800.0 PL=0
MOVL C01427 V=800.0 PL=0
MOVL C01428 V=800.0 PL=0
MOVL C01429 V=800.0 PL=0
MOVL C01430 V=800.0 PL=0
MOVL C01431 V=800.0 PL=0
MOVL C01432 V=800.0 PL=0
MOVL C01433 V=800.0 PL=0
MOVL C01434 V=800.0 PL=0
MOVL C01435 V=800.0 PL=0
MOVL C01436 V=800.0 PL=0
MOVL C01437 V=800.0 PL=0
MOVL C01438 V=800.0 PL=0
MOVL C01439 V=800.0 PL=0
MOVL C01440 V=800.0 PL=0
MOVL C01441 V=800.0 PL=0
MOVL C01442 V=800.0 PL=0
MOVL C01443 V=800.0 PL=0
MOVL C01444 V=800.0 PL=0
MOVL C01445 V=800.0 PL=0
MOVL C01446 V=800.0 PL=0
MOVL C01447 V=800.0 PL=0
MOVL C01448 V=800.0 PL=0
MOVL C01449 V=800.0 PL=0
MOVL C01450 V=800.0 PL=0
MOVL C01451 V=800.0 PL=0
MOVL C01452 V=800.0 PL=0
MOVL C01453 V=800.0 PL=0
MOVL C01454 V=800.0 PL=0
MOVL C01455 V=800.0 PL=0
MOVL C01456 V=800.0 PL=0
MOVL C01457 V=800.0 PL=0
MOVL C01458 V=800.0 PL=0
MOVL C01459 V=800.0 PL=0
MOVL C01460 V=800.0 PL=0
MOVL C01461 V=800.0 PL=0
MOVL C01462 V=800.0 PL=0
MOVL C01463 V=800.0 PL=0
MOVL C01464 V=800.0 PL=0
MOVL C01465 V=800.0 PL=0
MOVL C01466 V=800.0 PL=0
MOVL C01467 V=800.0 PL=0
MOVL C01468 V=800.0 PL=0
MOVL C01469 V=800.0 PL=0
MOVL C01470 V=800.0 PL=0
MOVL C01471 V=800.0 PL=0
MOVL C01472 V=800.0 PL=0
MOVL C01473 V=800.0 PL=0
MOVL C01474 V=800.0 PL=0
MOVL C01475 V=800.0 PL=0
MOVL C01476 V=800.0 PL=0
MOVL C01477 V=800.0 PL=0
MOVL C01478 V=800.0 PL=0
MOVL C01479 V=800.0 PL=0
MOVL C01480 V=800.0 PL=0
MOVL C01481 V=800.0 PL=0
MOVL C01482 V=800.0 PL=0
MOVL C01483 V=800.0 PL=0
MOVL C01484 V=800.0 PL=0
MOVL C01485 V=800.0 PL=0
MOVL C01486 V=800.0 PL=0
MOVL C01487 V=800.0 PL=0
MOVL C01488 V=800.0 PL=0
MOVL C01489 V=800.0 PL=0
MOVL C01490 V=800.0 PL=0
MOVL C01491 V=800.0 PL=0
MOVL C01492 V=800.0 PL=0
MOVL C01493 V=800.0 PL=0
MOVL C01494 V=800.0 PL=0
MOVL C01495 V=800.0 PL=0
MOVL C01496 V=800.0 PL=0
MOVL C01497 V=800.0 PL=0
MOVL C01498 V=800.0 PL=0
MOVL C01499 V=800.0 PL=0
MOVL C01500 V=800.0 PL=0
MOVL C01501 V=800.0 PL=0
MOVL C01502 V=800.0 PL=0
MOVL C01503 V=800.0 PL=0
MOVL C01504 V=800.0 PL=0
MOVL C01505 V=800.0 PL=0
MOVL C01506 V=800.0 PL=0
MOVL C01507 V=800.0 PL=0
MOVL C01508 V=800.0 PL=0
MOVL C01509 V=800.0 PL=0
MOVL C01510 V=800.0 PL=0
MOVL C01511 V=800.0 PL=0
MOVL C01512 V=800.0 PL=0
MOVL C01513 V=800.0 PL=0
MOVL C01514 V=800.0 PL=0
MOVL C01515 V=800.0 PL=0
MOVL C01516 V=800.0 PL=0
MOVL C01517 V=800.0 PL=0
MOVL C01518 V=800.0 PL=0
MOVL C01519 V=800.0 PL=0
MOVL C01520 V=800.0 PL=0
MOVL C01521 V=800.0 PL=0
MOVL C01522 V=800.0 PL=0
MOVL C01523 V=800.0 PL=0
MOVL C01524 V=800.0 PL=0
MOVL C01525 V=800.0 PL=0
MOVL C01526 V=800.0 PL=0
MOVL C01527 V=800.0 PL=0
MOVL C01528 V=800.0 PL=0
MOVL C01529 V=800.0 PL=0
MOVL C01530 V=800.0 PL=0
MOVL C01531 V=800.0 PL=0
MOVL C01532 V=800.0 PL=0
MOVL C01533 V=800.0 PL=0
MOVL C01534 V=800.0 PL=0
MOVL C01535 V=800.0 PL=0
MOVL C01536 V=800.0 PL=0
MOVL C01537 V=800.0 PL=0
MOVL C01538 V=800.0 PL=0
MOVL C01539 V=800.0 PL=0
MOVL C01540 V=800.0 PL=0
MOVL C01541 V=800.0 PL=0
MOVL C01542 V=800.0 PL=0
MOVL C01543 V=800.0 PL=0
MOVL C01544 V=800.0 PL=0
MOVL C01545 V=800.0 PL=0
MOVL C01546 V=800.0 PL=0
MOVL C01547 V=800.0 PL=0
MOVL C01548 V=800.0 PL=0
MOVL C01549 V=800.0 PL=0
MOVL C01550 V=800.0 PL=0
MOVL C01551 V=800.0 PL=0
MOVL C01552 V=800.0 PL=0
MOVL C01553 V=800.0 PL=0
MOVL C01554 V=800.0 PL=0
MOVL C01555 V=800.0 PL=0
MOVL C01556 V=800.0 PL=0
MOVL C01557 V=800.0 PL=0
MOVL C01558 V=800.0 PL=0
MOVL C01559 V=800.0 PL=0
MOVL C01560 V=800.0 PL=0
MOVL C01561 V=800.0 PL=0
MOVL C01562 V=800.0 PL=0
MOVL C01563 V=800.0 PL=0
MOVL C01564 V=800.0 PL=0
MOVL C01565 V=800.0 PL=0
MOVL C01566 V=800.0 PL=0
MOVL C01567 V=800.0 PL=0
MOVL C01568 V=800.0 PL=0
MOVL C01569 V=800.0 PL=0
MOVL C01570 V=800.0 PL=0
MOVL C01571 V=800.0 PL=0
MOVL C01572 V=800.0 PL=0
MOVL C01573 V=800.0 PL=0
MOVL C01574 V=800.0 PL=0
MOVL C01575 V=800.0 PL=0
MOVL C01576 V=800.0 PL=0
MOVL C01577 V=800.0 PL=0
MOVL C01578 V=800.0 PL=0
MOVL C01579 V=800.0 PL=0
MOVL C01580 V=800.0 PL=0
MOVL C01581 V=800.0 PL=0
MOVL C01582 V=800.0 PL=0
MOVL C01583 V=800.0 PL=0
MOVL C01584 V=800.0 PL=0
MOVL C01585 V=800.0 PL=0
MOVL C01586 V=800.0 PL=0
MOVL C01587 V=800.0 PL=0
MOVL C01588 V=800.0 PL=0
MOVL C01589 V=800.0 PL=0
MOVL C01590 V=800.0 PL=0
MOVL C01591 V=800.0 PL=0
MOVL C01592 V=800.0 PL=0
MOVL C01593 V=800.0 PL=0
MOVL C01594 V=800.0 PL=0
MOVL C01595 V=800.0 PL=0
MOVL C01596 V=800.0 PL=0
MOVL C01597 V=800.0 PL=0
MOVL C01598 V=800.0 PL=0
MOVL C01599 V=800.0 PL=0
MOVL C01600 V=800.0 PL=0
MOVL C01601 V=800.0 PL=0
MOVL C01602 V=800.0 PL=0
MOVL C01603 V=800.0 PL=0
MOVL C01604 V=800.0 PL=0
MOVL C01605 V=800.0 PL=0
MOVL C01606 V=800.0 PL=0
MOVL C01607 V=800.0 PL=0
MOVL C01608 V=800.0 PL=0
MOVL C01609 V=800.0 PL=0
MOVL C01610 V=800.0 PL=0
MOVL C01611 V=800.0 PL=0
MOVL C01612 V=800.0 PL=0
MOVL C01613 V=800.0 PL=0
MOVL C01614 V=800.0 PL=0
MOVL C01615 V=800.0 PL=0
MOVL C01616 V=800.0 PL=0
MOVL C01617 V=800.0 PL=0
MOVL C01618 V=800.0 PL=0
MOVL C01619 V=800.0 PL=0
MOVL C01620 V=800.0 PL=0
MOVL C01621 V=800.0 PL=0
MOVL C01622 V=800.0 PL=0
MOVL C01623 V=800.0 PL=0
MOVL C01624 V=800.0 PL=0
MOVL C01625 V=800.0 PL=0
